METHOD M_Activity_Stop_PTCs : BOOL
VAR_INPUT
END_VAR
VAR_INST
	
END_VAR

out_bStop_PTCs := TRUE;

logs.M_LogInfo('STOP all PTCs...');
	
	
stat.nState := E_MET_CRYO_WARMUP_STATE.START_RAMP_Up_DETECTORS_1K;
END_METHOD

METHOD M_Activity_Stopping_Warm_Up
VAR_INPUT
END_VAR
VAR_IN_OUT
	{attribute 'OPC.UA.DA' := '0'}
	all_cryo_temps:					FB_METIS_TEMPERATURES;
	{attribute 'OPC.UA.DA' := '0'}
	all_heaters:					FB_METIS_HEATERS;
	{attribute 'OPC.UA.DA' := '0'}
	all_t_ctrls:      				FB_METIS_TCTRL;
	{attribute 'OPC.UA.DA' := '0'}
	all_t_votes: 					FB_METIS_VOTERS;
	{attribute 'OPC.UA.DA' := '0'}
	interlocks:						T_METIS_CRYO_INTERLOCKS;
END_VAR
// TODO CRY VOTE 8 



	all_heaters.h_cry_sha.M_SetDisable();
	all_heaters.h_cry_shb.M_SetDisable();
	all_heaters.h_cry_shc.M_SetDisable();

	all_t_ctrls.tc_cry_sha.M_SetDisable();
	all_t_ctrls.tc_cry_shb.M_SetDisable();
	all_t_ctrls.tc_cry_shc.M_SetDisable();
	stat.nState := E_MET_CRYO_WARMUP_STATE.FINISHED;
	stat.sState := 'Stopping Warm Up...';
	
	logs.M_LogInfo('Stopping heaters and temperature controls...');
END_METHOD

METHOD M_AreWarmUpHeaterActive : BOOL
VAR_INPUT
END_VAR
END_METHOD

METHOD M_CheckTCErrors
VAR_INPUT
END_VAR
VAR_IN_OUT
	{attribute 'OPC.UA.DA' := '0'}
	all_cryo_temps:					FB_METIS_TEMPERATURES;
	{attribute 'OPC.UA.DA' := '0'}
	all_heaters:					FB_METIS_HEATERS;
	{attribute 'OPC.UA.DA' := '0'}
	all_t_ctrls:      				FB_METIS_TCTRL;
	{attribute 'OPC.UA.DA' := '0'}
	all_t_votes: 					FB_METIS_VOTERS;
	{attribute 'OPC.UA.DA' := '0'}
	interlocks:						T_METIS_CRYO_INTERLOCKS;
END_VAR
IF all_heaters.h_cry_sha.M_isHeaterInError() OR all_t_ctrls.tc_cry_sha.stat.bError THEN
	stat.bError := TRUE;
	//M_SetError(E8100_StiffRingTempCtrlError, 'ERROR: Stiff Ring temp control - Check the complete Control-loop');

END_IF

IF all_heaters.h_cry_shb.M_isHeaterInError() OR all_t_ctrls.tc_cry_shb.stat.bError THEN
	stat.bError := TRUE;
	//M_SetError(E8101_IntermediateSegmentTempCtrlError, 'ERROR: Intermediate segment temp control - Check the complete Control-loop');
END_IF

IF all_heaters.h_cry_shc.M_isHeaterInError() OR all_t_ctrls.tc_cry_shc.stat.bError THEN
	stat.bError := TRUE;
	//M_SetError(E8102_BottomSegmentTempCtrlError, 'ERROR: Bottom Segment - Check the complete Control-loop');

END_IF

IF (all_heaters.h_cry_sha.M_isHeaterInError() OR all_t_ctrls.tc_cry_sha.stat.bError) AND 
	(all_heaters.h_cry_shb.M_isHeaterInError() OR all_t_ctrls.tc_cry_shb.stat.bError) AND
	(all_heaters.h_cry_shc.M_isHeaterInError() OR all_t_ctrls.tc_cry_shc.stat.bError) THEN
	stat.bError := TRUE;
	//M_SetError(E8103_OneOrMoreTempCtrlInError, 'ERROR: One or more temp control - Check the Control-loop');
	RETURN;
END_IF
END_METHOD

METHOD M_Configure
VAR_INPUT
END_VAR
IF NOT stat.bConfigured THEN


// Event Handleing 

arrEventEntry[0] := Tc_Events.METIS_Cryo_Routine.Routine_Started;
arrEventEntry[1] := Tc_Events.METIS_Cryo_Routine.Routine_Stopped_Manually;
arrEventEntry[2] := Tc_Events.METIS_Cryo_Routine.Routine_Stopped_Automatically;
arrEventEntry[3] := Tc_Events.METIS_Cryo_Routine.Routine_Completed_Successfully;
arrEventEntry[4] := Tc_Events.METIS_Cryo_Routine.Routine_FailedToStart;
arrEventEntry[5] := Tc_Events.METIS_Cryo_Routine.Routine_Aborted_CriticalFault;
arrEventEntry[6] := Tc_Events.METIS_Cryo_Routine.Routine_Interlock_ConflictDetected;


//////


// This call just configures logs at the very start.
// Logging is done by explicit calls to M_LogInfo().
logs(in_sName := in_sName);



// A MUST !!!
stat.bConfigured	:= TRUE;


END_IF
END_METHOD

METHOD M_HandleEvents
VAR_INPUT
END_VAR

//
// Handle triggers
//

trigEnable	(CLK := ctrl.bEnable);
trigDisable	(CLK := ctrl.bEnable);

// Array of EventEntry is initialised in the M_Configure method with 
// the alarms defined for the Valve.

fbAlarmHandler(stAlarms := stAlarms);


// Set Alarms

IF trigEnable.Q	THEN
	fbAlarmHandler.M_SetAlarm(Tc_Events.METIS_Cryo_Routine.Routine_Started);
END_IF

IF trigDisable.Q	THEN
	fbAlarmHandler.M_SetAlarm(Tc_Events.METIS_Cryo_Routine.Routine_Stopped_Manually);
END_IF

IF stat.bDone THEN
	fbAlarmHandler.M_SetAlarm(Tc_Events.METIS_Cryo_Routine.Routine_Completed_Successfully);
END_IF

IF stat.bAlarm THEN
	fbAlarmHandler.M_SetAlarm(Tc_Events.METIS_Cryo_Routine.Routine_Aborted_CriticalFault);
	fbAlarmHandler.M_SetAlarm(Tc_Events.METIS_Cryo_Routine.Routine_Stopped_Automatically);
END_IF

IF stat.bError THEN
	fbAlarmHandler.M_SetAlarm(Tc_Events.METIS_Cryo_Routine.Routine_FailedToStart);
END_IF

// Clear Alarms

IF NOT stat.bAlarm THEN
	fbAlarmHandler.M_ClearAlarm(Tc_Events.METIS_Cryo_Routine.Routine_Aborted_CriticalFault);
	fbAlarmHandler.M_ClearAlarm(Tc_Events.METIS_Cryo_Routine.Routine_Stopped_Automatically);
END_IF

IF NOT stat.bError THEN
	fbAlarmHandler.M_ClearAlarm(Tc_Events.METIS_Cryo_Routine.Routine_FailedToStart);
END_IF
END_METHOD

METHOD M_HandleInterlocks
VAR_INPUT
END_VAR
VAR_IN_OUT
	{attribute 'OPC.UA.DA' := '0'}
	all_cryo_temps:					FB_METIS_TEMPERATURES;
	{attribute 'OPC.UA.DA' := '0'}
	all_heaters:					FB_METIS_HEATERS;
	{attribute 'OPC.UA.DA' := '0'}
	all_t_ctrls:      				FB_METIS_TCTRL;
	{attribute 'OPC.UA.DA' := '0'}
	all_t_votes: 					FB_METIS_VOTERS;
	{attribute 'OPC.UA.DA' := '0'}
	interlocks:						T_METIS_CRYO_INTERLOCKS;
END_VAR



//interlocks.bInterlock_Evacuation 		:= FALSE;
//interlocks.bInterlock_Venting 			:= TRUE; // Venting blocked
//interlocks.bInterlock_CoolDown 			:= TRUE; // Cool_Down, pre-cooling, LN2_filling blocked
//interlocks.bInterlock_WarmUp 			:= TRUE; // Warm_up Blocked
//interlocks.bInterlock_Regeneration 		:= FALSE;
//interlocks.bInterlock_AntiFogging 		:= FALSE;
//interlocks.bInterlock_PowerOutage 		:= FALSE;
//interlocks.bInterlock_StopPowerOutage	:= FALSE;

//interlocks.sInterlockState := 'RE_GENERATION Active';
END_METHOD

METHOD M_PermitEvacuationStop : BOOL
VAR_INPUT
END_VAR
M_PermitEvacuationStop := stat.bPermitEvacuationStop;
END_METHOD

METHOD M_PermitVenting : BOOL
VAR_INPUT
END_VAR
END_METHOD

METHOD PRIVATE M_SetError
VAR_INPUT
    nCode     : UDINT;
    sMessage  : STRING;
END_VAR


stat.Error.nCode := nCode;
stat.Error.sMessage := sMessage;
stat.bError := TRUE;
//stat.nState := E_MET_CRYO_WARMUP_STATE.ERROR;
END_METHOD

METHOD M_StateMachine
VAR_INPUT
END_VAR
VAR_IN_OUT
	{attribute 'OPC.UA.DA' := '0'}
	all_cryo_temps:					FB_METIS_TEMPERATURES;
	{attribute 'OPC.UA.DA' := '0'}
	all_heaters:					FB_METIS_HEATERS;
	{attribute 'OPC.UA.DA' := '0'}
	all_t_ctrls:      				FB_METIS_TCTRL;
	{attribute 'OPC.UA.DA' := '0'}
	all_t_votes: 					FB_METIS_VOTERS;
	{attribute 'OPC.UA.DA' := '0'}
	interlocks:						T_METIS_CRYO_INTERLOCKS;
END_VAR


//--- State Machine Logic ---
CASE stat.nState OF
	
	E_MET_CRYO_WARMUP_STATE.NONE:
		
		M_Activity_None(interlocks := interlocks);
 
	E_MET_CRYO_WARMUP_STATE.CHECK_PRECONDITIONS:
	
		M_Activity_Check_Preconditions(); 
	
	E_MET_CRYO_WARMUP_STATE.START_WARM_UP:
	
		M_Activity_Start_Warm_Up();
		
	E_MET_CRYO_WARMUP_STATE.STOP_PTCs:
	
		M_Activity_Stop_PTCs();
 	
	E_MET_CRYO_WARMUP_STATE.START_RAMP_Up_DETECTORS_1K:
	
		M_Activity_Start_Ramp_Up_Detectors_1k();
	
	E_MET_CRYO_WARMUP_STATE.KEEP_RAMPING_Up_DETECTORS:
	
		M_Activity_Keep_Ramping_Up_Detectors();
	
	E_MET_CRYO_WARMUP_STATE.RAMP_UP_DETECTORS_6K:
	
		M_Activity_Ramp_Up_Detectors_2();
	
	E_MET_CRYO_WARMUP_STATE.START_RAMP_Up_RADIATION_SHIELDS:
	
		M_Activity_Start_Ramp_Up_Radiation_Shields(		
						all_cryo_temps:= all_cryo_temps,
						all_heaters := all_heaters,
						all_t_ctrls := all_t_ctrls,
						all_t_votes := all_t_votes,
						interlocks := interlocks);
		M_CheckTCErrors(all_cryo_temps:= all_cryo_temps,
						all_heaters := all_heaters,
						all_t_ctrls := all_t_ctrls,
						all_t_votes := all_t_votes,
						interlocks := interlocks);
	
	E_MET_CRYO_WARMUP_STATE.START_RAMP_Up_IMG:
	
		M_Activity_Start_Ramp_Up_IMG();
	
	E_MET_CRYO_WARMUP_STATE.START_RAMP_Up_SCAO:
	
		M_Activity_Start_Ramp_Up_SCAO();
	
	E_MET_CRYO_WARMUP_STATE.START_RAMP_Up_LMS:
	
		M_Activity_Start_Ramp_Up_LMS();
	
	E_MET_CRYO_WARMUP_STATE.START_RAMP_Up_CFO:
	
		M_Activity_Start_Ramp_Up_CFO();
	
	E_MET_CRYO_WARMUP_STATE.KEEP_WARMING_UP:
	
		M_Activity_Keep_Warming_Up(all_cryo_temps:= all_cryo_temps);
		
		M_CheckTCErrors(all_cryo_temps:= all_cryo_temps,
						all_heaters := all_heaters,
						all_t_ctrls := all_t_ctrls,
						all_t_votes := all_t_votes,
						interlocks := interlocks);
	
	E_MET_CRYO_WARMUP_STATE.STOPPING_WARM_UP:
	
		M_Activity_Stopping_Warm_Up(all_cryo_temps:= all_cryo_temps,
						all_heaters := all_heaters,
						all_t_ctrls := all_t_ctrls,
						all_t_votes := all_t_votes,
						interlocks := interlocks);
	
	E_MET_CRYO_WARMUP_STATE.FINISHED:
	
		M_Activity_Finished(); 
	
	E_MET_CRYO_WARMUP_STATE.ERROR:
	
		M_Activity_Error_Handling(all_cryo_temps:= all_cryo_temps,
						all_heaters := all_heaters,
						all_t_ctrls := all_t_ctrls,
						all_t_votes := all_t_votes,
						interlocks := interlocks);

END_CASE;
END_METHOD

METHOD M_UpdateStatus
VAR_INPUT
END_VAR


IF stat.nState = E_MET_CRYO_WARMUP_STATE.ERROR THEN
	stat.bError := TRUE;
ELSE
	stat.bError := FALSE;
END_IF



out_bWarmUpActive := stat.bActive;


// Check Pre-Conditions for HMI Enable 


stat.bPreConditionsMet := 	in_Cryo_Stat.bPumpsAreRunning 		AND
							in_Cryo_Stat.bEvacuationActive   	AND
							NOT in_Cryo_Stat.bCoolDownActive    AND
							in_Cryo_Stat.bVentingValvesAreClosed;
END_METHOD

END_FUNCTION_BLOCK

// POUs/Routines/Regeneration/FB_METIS_CRYO_REGENERATION
FUNCTION_BLOCK FB_METIS_CRYO_REGENERATION
VAR_INPUT
	in_sName:								STRING := 'RE-GENERATION';
	in_Cryo_Stat:							T_METIS_CRYO_STAT;
	in_lrRegeneration_Safe_Temp:			LREAL := 280.0;
	in_lrRegeneration_Safe_Press:			LREAL := 0.01;
    in_lrTemp_Regeneration_SetPoint: 		LREAL := 333.0;
    in_lrTemp_Regeneration_Alarm:			LREAL := 340.0;
    in_lrTemp_Regeneration_Stop:			LREAL := 310.0;
    in_tSorption_Pump_Cool_Down_TimeOut: 	TIME  := T#3H; 
END_VAR
VAR_OUTPUT
	out_bRegenerationActive : BOOL := FALSE; // TRUE when regeneration is active
END_VAR

VAR_IN_OUT
	{attribute 'OPC.UA.DA' := '0'}
	all_cryo_temps:					FB_METIS_TEMPERATURES;
	{attribute 'OPC.UA.DA' := '0'}
	all_heaters:					FB_METIS_HEATERS;
	{attribute 'OPC.UA.DA' := '0'}
	all_t_ctrls:      				FB_METIS_TCTRL;
	{attribute 'OPC.UA.DA' := '0'}
	all_t_votes: 					FB_METIS_VOTERS;
	{attribute 'OPC.UA.DA' := '0'}
	interlocks:						T_METIS_CRYO_INTERLOCKS;
END_VAR
VAR	
	t_vote_tc_cry_sp:				FB_METIS_VOTER;
	tc_sorption_pump:				FB_PWM_PID_CTRL;
	h_sorption_pump_heater:			FB_HEATER_PWM;		// 3.4 A terminal
	
	stat:							T_MET_CRYO_RE_GENERATION_STAT;
	ctrl:							T_MET_CRYO_RE_GENERATION_CTRL;


	
	bTest_run: BOOL := FALSE;
	
		// Triggers.
	//
	// Capture Enable/Disable.
	trigEnable:		R_TRIG;	// in_bEnable
	trigDisable:	F_TRIG;	// in_bEnable
	
	/////////////////////
	// Cryo System logs
	/////////////////////
		
	logs:	FB_CRYO_FUNCTION_LOG;
	
	// timeouts
	
	tonHeatingTimer     : TON;         // Timer to track the 3-hour heating period
	tHeatingTime:		TIME;
	lrHeatingTime:		LREAL := 3.0; // hours
	
	CoolDownTimeout:		TON;
	tCoolDownTime:			TIME;
	lrCoolDownTime:			LREAL := 1.0; // hours
	
	
END_VAR
VAR CONSTANT

    // --- [2000] Preconditions ---
    E2000_TemperaturesTooLow                      : UDINT := 2000001; // One or more cryostat temperatures < 280 K
    E2001_EvacuationNotActive                     : UDINT := 2000002; // Evacuation system not active
    E2002_RegenerationAlreadyRunning              : UDINT := 2000003; // Regeneration requested while already active
    E2003_CryostatPressureTooHigh_PreStart        : UDINT := 2000004; // Cryostat pressure > 1e-2 mbar before regeneration

    // --- [2100] Heater / Temperature Control Errors ---
    E2100_SorptionHeaterNotEnabled                : UDINT := 2100001; // Sorption pump heater failed to enable
    E2101_SorptionHeaterControlNotStarted         : UDINT := 2100002; // Temperature control did not start
    E2102_SorptionHeaterFailure                   : UDINT := 2100003; // Sorption pump heater failure detected
    E2103_SorptionHeaterShutdownFailure           : UDINT := 2100004; // Heater did not stop after regeneration

    // --- [2200] Temperature Monitoring Errors ---
    E2200_SP_TemperatureSensorFault               : UDINT := 2200001; // Sorption pump temperature sensor invalid
    E2201_SP_TemperatureNotRising                 : UDINT := 2200002; // Temperature not increasing during heating
    E2202_SP_TemperatureTooHigh                   : UDINT := 2200003; // Sorption pump temperature > 340 K
    E2203_SP_TemperatureNotCooling                : UDINT := 2200004; // Sorption pump not cooling after heater shutdown
    E2204_SP_CooldownTimeout                      : UDINT := 2200005; // Sorption pump cooldown timeout exceeded

    // --- [2300] Pressure Monitoring Errors ---
    E2300_CryostatPressureTooHigh                 : UDINT := 2300001; // Cryostat pressure > 1e-2 mbar during regeneration
    E2301_CryostatPressureRiseUnexpected          : UDINT := 2300002; // Unexpected pressure increase detected

    // --- [2400] Sequence Timing Errors ---
    E2400_RegenerationHeatingTimeout              : UDINT := 2400001; // Temperature did not reach target within allowed time
    E2401_RegenerationHoldTimeNotCompleted        : UDINT := 2400002; // 3-hour heating hold interrupted
    E2402_RegenerationSequenceTimeout             : UDINT := 2400003; // Regeneration procedure exceeded maximum duration

    // --- [2500] Manual Intervention ---
    E2500_OperatorStoppedRegeneration             : UDINT := 2500001; // Operator manually stopped regeneration
    E2501_OperatorDisabledHeater                  : UDINT := 2500002; // Heater disabled manually during regeneration

    // --- [2600] Interlock Violations ---
    E2600_LN2FillingActiveDuringRegeneration      : UDINT := 2600001; // Vessel filling active during regeneration
    E2601_PrecoolingActiveDuringRegeneration      : UDINT := 2600002; // Precooling system active during regeneration
    E2602_VentingActiveDuringRegeneration         : UDINT := 2600003; // Venting active during regeneration
    E2603_CoolingActiveDuringRegeneration         : UDINT := 2600004; // Cooling routine active during regeneration

    // --- [2700] Shutdown / Recovery Failures ---
    E2700_HeaterDidNotDisable                     : UDINT := 2700001; // Heater failed to disable during shutdown
    E2701_TemperatureControlDidNotStop            : UDINT := 2700002; // Temperature control still active after stop command
    E2702_RegenerationShutdownTimeout             : UDINT := 2700003; // Regeneration shutdown timeout exceeded

END_VAR


(*
	TODO: One of the initial conditions checks the minimum temperatures in the cryostat.
	The is still an open question to how to determine that.
	For time being with empty cryostat, a temperature on the Cryo body is considered to check the 
	minimum temperature 
*)

M_Configure();

M_HandleEvents();

M_ExecuteControllers();

M_StateMachine( 
	all_cryo_temps:= 							all_cryo_temps, 
	all_heaters:= 								all_heaters, 
	all_t_ctrls:= 								all_t_ctrls, 
	all_t_votes:=								all_t_votes, 
	interlocks:= 								interlocks);

M_UpdateStatus();



tHeatingTime := LREAL_TO_TIME(lrHeatingTime *  3600000.0);
tCoolDownTime := LREAL_TO_TIME(lrCoolDownTime * 3600000.0);

(* Re-Generation *)
METHOD M_Activity_Check_Preconditions : BOOL
VAR_INPUT
END_VAR
VAR_IN_OUT
	{attribute 'OPC.UA.DA' := '0'}
	all_cryo_temps:					FB_METIS_TEMPERATURES;
	{attribute 'OPC.UA.DA' := '0'}
	all_heaters:					FB_METIS_HEATERS;
	{attribute 'OPC.UA.DA' := '0'}
	all_t_ctrls:      				FB_METIS_TCTRL;
	{attribute 'OPC.UA.DA' := '0'}
	all_t_votes: 					FB_METIS_VOTERS;
	{attribute 'OPC.UA.DA' := '0'}
	interlocks:						T_METIS_CRYO_INTERLOCKS;
END_VAR


//  Precondition Check: Cryo Temperature validity
IF NOT in_Cryo_Stat.bLowestTempValid THEN
	//M_SetError(nCode := E3101_REGEN_INVALID_TEMP,
	//			sMessage := 'Error: Invalid lowest cryo temperature reading.');
	stat.sRecoverySuggestion := '';
	RETURN; 
END_IF

//  Precondition Check: Regeneration safe Temperature 
IF in_Cryo_Stat.lrLowestTempK <= in_lrRegeneration_Safe_Temp THEN

	stat.sState := 'Error: temperature is below the safe Regeneration temperature.';
	//M_SetError(nCode := E3107_REGEN_SYSTEM_BELOW_SAFE_REGEN,
	//			sMessage := 'Error: system temperature is below the safe Regeneration temp.');
	stat.sRecoverySuggestion := '';
	RETURN; // Exit this state
END_IF


//  Precondition Check: Evacuation Status 
IF NOT in_Cryo_Stat.bEvacuationActive THEN

	stat.nState := E_MET_CRYO_RE_GENERATION_STATE.CHECK_PRECONDITIONS;
	///M_SetError(nCode := E3108_REGEN_EVACUATION_NOT_ACTIVE,
	//			sMessage := 'Error: Evacuation not Active');
		stat.sRecoverySuggestion := 'Start Evacuation';			
	stat.bPermitEvacuationStop := FALSE; // Prevent premature stop of evacuation
	RETURN; // Exit this state until evacuation is active
END_IF

{IF defined (V1_HW)}

//  Precondition Check: Evacuation Status 
IF NOT in_Cryo_Stat.bRoughingPumpsAreRunning THEN

	stat.nState := E_MET_CRYO_RE_GENERATION_STATE.CHECK_PRECONDITIONS;
	M_SetError(nCode := E3106_REGEN_PUMPS_NOT_ACTIVE,
				sMessage := 'Error: One or both roughing pumps are not running');
		stat.sRecoverySuggestion := 'Start roughing pumps';			
	stat.bPermitEvacuationStop := FALSE; // Prevent premature stop of evacuation
	RETURN; // Exit this state until evacuation is active
	
ELSE
	
		;
END_IF

{END_IF}

stat.bActive := TRUE;
stat.bBusy 	 := TRUE;
stat.bDone   := FALSE;

// If all preconditions are met, proceed to the next state
stat.nState := E_MET_CRYO_RE_GENERATION_STATE.START_HEATING;

stat.sState := 'Regenerating...';
logs.M_LogInfo('Regeneration Started...');
END_METHOD

METHOD M_Activity_CoolDownSP : BOOL
VAR_INPUT
END_VAR
VAR_IN_OUT
	{attribute 'OPC.UA.DA' := '0'}
	all_cryo_temps:					FB_METIS_TEMPERATURES;
	{attribute 'OPC.UA.DA' := '0'}
	all_heaters:					FB_METIS_HEATERS;
	{attribute 'OPC.UA.DA' := '0'}
	all_t_ctrls:      				FB_METIS_TCTRL;
	{attribute 'OPC.UA.DA' := '0'}
	all_t_votes: 					FB_METIS_VOTERS;
	{attribute 'OPC.UA.DA' := '0'}
	interlocks:						T_METIS_CRYO_INTERLOCKS;
END_VAR
	all_heaters.h_cry_sp.M_SetDisable();
	all_t_ctrls.tc_cry_sp.M_SetDisable();
	tonHeatingTimer(IN:=FALSE); // Reset Timer
	
	IF all_cryo_temps.t_cry_vot_10.stat.lrTempK < in_lrTemp_Regeneration_Stop THEN
		stat.nState := E_MET_CRYO_RE_GENERATION_STATE.FINISHED;
		cooldownTimeout(IN := FALSE);
	ELSE
		stat.nState := E_MET_CRYO_RE_GENERATION_STATE.COOL_DOWN;
		stat.sState := 'Sorption-pump cooling down';
	END_IF
	
	cooldownTimeout(IN := TRUE, PT := tCoolDownTime);
	stat.sState :=  CONCAT('Sorption-pump cooling down...', F_TON_TO_TIME_STRING(Timer := cooldownTimeout));

	IF cooldownTimeout.Q THEN
		logs.M_LogWarning('Cooldown timeout. Sorption pump did not cool sufficiently.');
		cooldownTimeout(IN := FALSE);
		//stat.nState := E_MET_CRYO_RE_GENERATION_STATE.ERROR;
		RETURN;
	END_IF
END_METHOD

METHOD M_Activity_ErrorHandeling : BOOL
VAR_INPUT
END_VAR
VAR_IN_OUT
	{attribute 'OPC.UA.DA' := '0'}
	all_cryo_temps:					FB_METIS_TEMPERATURES;
	{attribute 'OPC.UA.DA' := '0'}
	all_heaters:					FB_METIS_HEATERS;
	{attribute 'OPC.UA.DA' := '0'}
	all_t_ctrls:      				FB_METIS_TCTRL;
	{attribute 'OPC.UA.DA' := '0'}
	all_t_votes: 					FB_METIS_VOTERS;
	{attribute 'OPC.UA.DA' := '0'}
	interlocks:						T_METIS_CRYO_INTERLOCKS;
END_VAR
        stat.bActive := TRUE;
        in_cryo_stat.bPermitEvacuationStop := FALSE; // Evacuation cannot stop, yet
		all_heaters.h_cry_sp.M_SetDisable();
		all_t_ctrls.tc_cry_sp.M_SetDisable();
        
		IF all_cryo_temps.t_cry_vot_10.stat.lrTempK < in_lrTemp_Regeneration_Stop THEN
            stat.nState := E_MET_CRYO_RE_GENERATION_STATE.NONE;
			stat.bActive := FALSE;
			stat.bBusy := FALSE;
			ctrl.bEnable := FALSE;						// Disable Regeneration
			stat.bPermitEvacuationStop := TRUE; // Evacuation can stop
		ELSE
			stat.nState := E_MET_CRYO_RE_GENERATION_STATE.COOL_DOWN;
			stat.sState := 'Sorption-pump cooling down';
        END_IF
		
        IF ctrl.bReset THEN
			logs.M_LogInfo('Reset received. Restarting regeneration.'); 
            stat.nState := E_MET_CRYO_RE_GENERATION_STATE.NONE;
			ctrl.bReset := FALSE;
			ctrl.bEnable := FALSE;						// Disable Regeneration
        END_IF
END_METHOD

METHOD M_Activity_Finished : BOOL
VAR_INPUT
END_VAR
VAR_IN_OUT
	{attribute 'OPC.UA.DA' := '0'}
	all_cryo_temps:					FB_METIS_TEMPERATURES;
	{attribute 'OPC.UA.DA' := '0'}
	all_heaters:					FB_METIS_HEATERS;
	{attribute 'OPC.UA.DA' := '0'}
	all_t_ctrls:      				FB_METIS_TCTRL;
	{attribute 'OPC.UA.DA' := '0'}
	all_t_votes: 					FB_METIS_VOTERS;
	{attribute 'OPC.UA.DA' := '0'}
	interlocks:						T_METIS_CRYO_INTERLOCKS;
END_VAR


//stat.bPermitEvacuationStop := TRUE; // Evacuation can stop
all_heaters.h_cry_sp.M_SetDisable();
all_t_ctrls.tc_cry_sp.M_SetDisable();
stat.sState := 'Re_generation finished';
tonHeatingTimer.IN := FALSE; // Reset Timer
	
ctrl.bEnable := FALSE;			// Disable Regeneration

stat.nState := E_MET_CRYO_RE_GENERATION_STATE.NONE;
logs.M_LogInfo('Sorption regeneration finished.');

stat.bActive := FALSE;
stat.bBusy 	 := FALSE;
stat.bDone   := TRUE;

cooldownTimeout(IN := FALSE);
tonHeatingTimer(IN := FALSE);
END_METHOD

METHOD M_Activity_KeepHeating : BOOL
VAR_INPUT
END_VAR
VAR_IN_OUT
    {attribute 'OPC.UA.DA' := '0'}
    all_cryo_temps : FB_METIS_TEMPERATURES;
    {attribute 'OPC.UA.DA' := '0'}
    all_heaters    : FB_METIS_HEATERS;
    {attribute 'OPC.UA.DA' := '0'}
    all_t_ctrls    : FB_METIS_TCTRL;
    {attribute 'OPC.UA.DA' := '0'}
    all_t_votes    : FB_METIS_VOTERS;
    {attribute 'OPC.UA.DA' := '0'}
    interlocks     : T_METIS_CRYO_INTERLOCKS;
END_VAR
VAR_INST
    nHeatingState  : UINT := 0;
    bLoggedReached : BOOL := FALSE;
	
	tonTempSenseGlitch : TON;                 // 3 minute grace window
    bTempSenseGlitchActive : BOOL := FALSE;   // latched while in grace window
END_VAR
VAR
    lrTempK        : LREAL;
    bHeaterError   : BOOL;
    bOverTemp      : BOOL;
    bDisableReq    : BOOL;

    bTempGlitchNow  : BOOL;
END_VAR
M_Activity_KeepHeating := FALSE;

// Snapshot values
lrTempK      := all_cryo_temps.t_cry_vot_10.stat.lrTempK;
bHeaterError := all_heaters.h_cry_sp.M_isHeaterInError();
bDisableReq  := trigDisable.Q;

////////////////////////////////////////////////////
// Temp Sensor glitch handling: lrTempK forced to >900K
////////////////////////////////////////////////////
bTempGlitchNow := (lrTempK > 900.0);

// Start / run 3-minute grace timer while glitch is present
IF bTempGlitchNow THEN
    bTempSenseGlitchActive := TRUE;
    tonTempSenseGlitch(IN := TRUE, PT := T#3M);

ELSE
    // Glitch not present now
    IF bTempSenseGlitchActive THEN
        // We were in a glitch window and it recovered before timing out
        IF NOT tonTempSenseGlitch.Q THEN
            //M_SetError(E3000_REGEN_ERROR_CLEARED, '');
            stat.sRecoverySuggestion := '';
        END_IF

        // Stop and reset the glitch timer/window
        bTempSenseGlitchActive := FALSE;
        tonTempSenseGlitch(IN := FALSE, PT := T#3M);
    ELSE
        // Ensure timer is reset if not used
        tonTempSenseGlitch(IN := FALSE, PT := T#3M);
    END_IF
END_IF

// If glitch persists beyond 3 minutes, we stop masking.
// From that moment onward, the normal over-temperature check may act.
IF bTempSenseGlitchActive AND tonTempSenseGlitch.Q THEN
    // Grace window expired -> stop masking further
    bTempSenseGlitchActive := FALSE;
    tonTempSenseGlitch(IN := FALSE, PT := T#3M);
END_IF

//////////////////////////////////////////
// operator interrupt / errors
/////////////////////////////////////////

// Operator interrupt
IF bDisableReq THEN
    stat.sState := 'REGENERATION interrupted by the operator...';
    logs.M_LogInfo('REGENERATION interrupted by the operator...');
    stat.nState := E_MET_CRYO_RE_GENERATION_STATE.COOL_DOWN;

    all_heaters.h_cry_sp.M_SetDisable();
    all_t_ctrls.tc_cry_sp.M_SetDisable();
    tonHeatingTimer(IN := FALSE);
    cooldownTimeout(IN := FALSE);

    // Reset internal state
    nHeatingState := 0;
    bLoggedReached := FALSE;

    // Reset EMI logic state too
    bTempSenseGlitchActive := FALSE;
    tonTempSenseGlitch(IN := FALSE, PT := T#3M);

    RETURN;
END_IF

// Over-temperature alarm: take action immediately,
// BUT only if we are NOT currently masking due to Temp Sensor glitch grace window.
bOverTemp := (lrTempK > in_lrTemp_Regeneration_Alarm);

IF bOverTemp AND (NOT bTempSenseGlitchActive) THEN
    logs.M_LogWarning('Temperature exceeds safe limit!');
    //M_SetError(E3102_REGEN_OVER_TEMP, 'Temperature at SP above alarm limit');
    stat.bAlarm := TRUE;

    stat.nState := E_MET_CRYO_RE_GENERATION_STATE.COOL_DOWN;
    stat.sState := 'Alarm: Sorption pump overheated';

    all_heaters.h_cry_sp.M_SetDisable();
    all_t_ctrls.tc_cry_sp.M_SetDisable();
    tonHeatingTimer(IN := FALSE);
    cooldownTimeout(IN := FALSE);

    // Reset internal state
    nHeatingState := 0;
    bLoggedReached := FALSE;

    // Reset Glitch logic state too
    bTempSenseGlitchActive := FALSE;
    tonTempSenseGlitch(IN := FALSE, PT := T#3M);

    RETURN;
END_IF

// Heater error 
IF all_heaters.h_cry_sp.M_isHeaterInError() THEN
{IF defined (V1_HW)}
 //   stat.nState := E_MET_CRYO_RE_GENERATION_STATE.COOL_DOWN;
    logs.M_LogInfo('SP heater failed, Regeneration stopped.');
    stat.sState := 'Heater error';
    M_SetError(E3105_REGEN_HEATER_FAIL, 'Heater at SP failed');
    stat.sRecoverySuggestion := 'Check SP heater controller';

//    all_heaters.h_cry_sp.M_SetDisable();
//    all_t_ctrls.tc_cry_sp.M_SetDisable();
//    tonHeatingTimer(IN := FALSE);
//    cooldownTimeout(IN := FALSE);

//    // Reset internal state
//    nHeatingState := 0;
//    bLoggedReached := FALSE;

//    // Reset Glitch logic state too
//    bTempSenseGlitchActive := FALSE;
//    tonTempSenseGlitch(IN := FALSE, PT := T#3M);

    RETURN;
{END_IF}
END_IF

/////////////////////////////////////////////////////
// state machine (normal operation)
/////////////////////////////////////////////////////
CASE nHeatingState OF
    0:
        in_cryo_stat.sState := 'REGENERATION Active';
        stat.sState := CONCAT('Sorption pump heating up to ',
                       CONCAT(LREAL_TO_STRING(in_lrTemp_Regeneration_SetPoint), ' K'));

        tonHeatingTimer(IN := FALSE);

        IF lrTempK >= in_lrTemp_Regeneration_SetPoint THEN
            nHeatingState := 10;
            bLoggedReached := FALSE;
        END_IF

    10:
        IF NOT bLoggedReached THEN
            logs.M_LogInfo(CONCAT(LREAL_TO_STRING(in_lrTemp_Regeneration_SetPoint), ' K achieved at Sorption Pump'));
            bLoggedReached := TRUE;
        END_IF

        tonHeatingTimer(IN := TRUE, PT := tHeatingTime);

        stat.sState := CONCAT(
            'Sorption pump heating hold... ',
            F_TON_TO_TIME_STRING(Timer := tonHeatingTimer)
        );

        IF tonHeatingTimer.Q THEN
            tonHeatingTimer(IN := FALSE);
            nHeatingState := 20;
        END_IF

    20:
        stat.nState := E_MET_CRYO_RE_GENERATION_STATE.COOL_DOWN;
        stat.sState := 'Transition: heating duration completed';
        logs.M_LogWarning('Transition: heating duration completed');
        nHeatingState := 99;

    99:
        tonHeatingTimer(IN := FALSE);
        cooldownTimeout(IN := FALSE);
        nHeatingState := 0;
        bLoggedReached := FALSE;

    ELSE
        tonHeatingTimer(IN := FALSE);
        cooldownTimeout(IN := FALSE);
        nHeatingState := 0;
        bLoggedReached := FALSE;
END_CASE
END_METHOD

METHOD M_Activity_None : BOOL
VAR_INPUT
END_VAR
VAR_IN_OUT
	{attribute 'OPC.UA.DA' := '0'}
	all_cryo_temps:					FB_METIS_TEMPERATURES;
	{attribute 'OPC.UA.DA' := '0'}
	all_heaters:					FB_METIS_HEATERS;
	{attribute 'OPC.UA.DA' := '0'}
	all_t_ctrls:      				FB_METIS_TCTRL;
	{attribute 'OPC.UA.DA' := '0'}
	all_t_votes: 					FB_METIS_VOTERS;
	{attribute 'OPC.UA.DA' := '0'}
	interlocks:						T_METIS_CRYO_INTERLOCKS;
END_VAR
stat.bActive := FALSE;
stat.bBusy := FALSE;
stat.bDone := TRUE;
stat.bReadyToDisable := FALSE;
stat.bPermitEvacuationStop := FALSE; // Evacuation is not allowed to stop
tonHeatingTimer(IN:=FALSE, PT:= tHeatingTime);
cooldownTimeout(IN := FALSE);


IF ctrl.bEnable AND NOT interlocks.bInterlock_Regeneration THEN  // Check interlocks
	stat.nState := E_MET_CRYO_RE_GENERATION_STATE.CHECK_PRECONDITIONS;
	stat.sState := 'Starting...Checking Preconditions';
	logs.M_LogInfo('REGENERATION started by the operator...Checking Preconditions');
ELSE
	stat.nState := E_MET_CRYO_RE_GENERATION_STATE.NONE;
	stat.sState := 'Re_generation OFF';
END_IF
END_METHOD

METHOD M_Activity_StartHeating : BOOL
VAR_INPUT
END_VAR
VAR_IN_OUT
	{attribute 'OPC.UA.DA' := '0'}
	all_cryo_temps:					FB_METIS_TEMPERATURES;
	{attribute 'OPC.UA.DA' := '0'}
	all_heaters:					FB_METIS_HEATERS;
	{attribute 'OPC.UA.DA' := '0'}
	all_t_ctrls:      				FB_METIS_TCTRL;
	{attribute 'OPC.UA.DA' := '0'}
	all_t_votes: 					FB_METIS_VOTERS;
	{attribute 'OPC.UA.DA' := '0'}
	interlocks:						T_METIS_CRYO_INTERLOCKS;
END_VAR
        stat.bActive := TRUE;
		in_cryo_stat.sState := 'RE_GENERATION Active';
		
		stat.bPermitEvacuationStop := FALSE; // Evacuation is not allowed to stop
		
		// Enable SP Heater
		all_heaters.h_cry_sp.M_SetEnable();
		
		all_t_ctrls.tc_cry_sp.M_SetEnable();
		
		all_t_ctrls.tc_cry_sp.M_Set_SetPoint(
			m_eSetpointType := E_METIS_CTRL_SETPOINT_SWITCH.FIXED,
			m_lrFixedSetpoint := in_lrTemp_Regeneration_SetPoint,
			m_lrSetpointOffset := 0.0, 
			m_pSetpointTemp := all_cryo_temps.M_SetTemperatureSensor(0));
			
        tonHeatingTimer(IN:=TRUE, PT:= tHeatingTime);
		
        stat.nState := E_MET_CRYO_RE_GENERATION_STATE.KEEP_HEATING;
END_METHOD

METHOD M_Configure
VAR_INPUT
END_VAR

IF NOT stat.bConfigured THEN
	

// This call just configures logs at the very start.
// Logging is done by explicit calls to M_LogInfo().
logs(in_sName := in_sName);


stat.bConfigured := TRUE;

END_IF
END_METHOD

METHOD M_ExecuteControllers
VAR_INPUT
END_VAR





//h_sorption_pump_heater(in_sName:= , in_fHeaterResistance:= , in_nMaxHeaterPower:= , in_HeaterCtrlType:= );

//t_vote_tc_cry_sp(
//		in_sName:= 't_vote_tc_cry_sp', 
//		in_bSimulation:= FALSE, 
//		in_nRampPeriodSec:= 10, 
//		met_temp:= all_cryo_temps);
		
//tc_sorption_pump(
//	in_sName:= 'tc_sorption_pump',
//	in_bEnable:= ctrl.bEnable_Temp_Ctrl, 
//	in_lrSetPoint:= lrTemp_Regeneration_SetPoint,
//	heater:= h_sorption_pump_heater,
//	temperature:= t_vote_tc_cry_sp);
END_METHOD

METHOD M_HandleEvents
VAR_INPUT
END_VAR

//
// Handle triggers
//

trigEnable	(CLK := ctrl.bEnable);
trigDisable	(CLK := ctrl.bEnable);
END_METHOD

METHOD M_PermitEvacuationStop : BOOL
VAR_INPUT
END_VAR
M_PermitEvacuationStop := stat.bPermitEvacuationStop;
END_METHOD

METHOD PRIVATE M_SetError
VAR_INPUT
    nCode     : UDINT;
    sMessage  : STRING;
END_VAR


stat.Error.nCode := nCode;
stat.Error.sMessage := sMessage;
stat.bError := TRUE;
//stat.nState := E_MET_CRYO_RE_GENERATION_STATE.ERROR;
END_METHOD

METHOD M_StateMachine
VAR_INPUT
	
END_VAR
VAR_IN_OUT
	{attribute 'OPC.UA.DA' := '0'}
	all_cryo_temps:					FB_METIS_TEMPERATURES;
	{attribute 'OPC.UA.DA' := '0'}
	all_heaters:					FB_METIS_HEATERS;
	{attribute 'OPC.UA.DA' := '0'}
	all_t_ctrls:      				FB_METIS_TCTRL;
	{attribute 'OPC.UA.DA' := '0'}
	all_t_votes: 					FB_METIS_VOTERS;
	{attribute 'OPC.UA.DA' := '0'}
	interlocks:						T_METIS_CRYO_INTERLOCKS;
END_VAR
VAR_INST
		

END_VAR

CASE stat.nState OF
    E_MET_CRYO_RE_GENERATION_STATE.NONE:
	
		M_Activity_None(
				all_cryo_temps:= all_cryo_temps,
				all_heaters := all_heaters,
				all_t_ctrls := all_t_ctrls,
				all_t_votes := all_t_votes,
				interlocks := interlocks);

    E_MET_CRYO_RE_GENERATION_STATE.CHECK_PRECONDITIONS:

		M_Activity_Check_Preconditions(
				all_cryo_temps:= all_cryo_temps,
				all_heaters := all_heaters,
				all_t_ctrls := all_t_ctrls,
				all_t_votes := all_t_votes,
				interlocks := interlocks);
		
    E_MET_CRYO_RE_GENERATION_STATE.START_HEATING:
	
		M_Activity_StartHeating(
				all_cryo_temps:= all_cryo_temps,
				all_heaters := all_heaters,
				all_t_ctrls := all_t_ctrls,
				all_t_votes := all_t_votes,
				interlocks := interlocks);

	E_MET_CRYO_RE_GENERATION_STATE.KEEP_HEATING:
	
		M_Activity_KeepHeating(
				all_cryo_temps:= all_cryo_temps,
				all_heaters := all_heaters,
				all_t_ctrls := all_t_ctrls,
				all_t_votes := all_t_votes,
				interlocks := interlocks);
		
    E_MET_CRYO_RE_GENERATION_STATE.COOL_DOWN:
	
		M_Activity_CoolDownSP(
				all_cryo_temps:= all_cryo_temps,
				all_heaters := all_heaters,
				all_t_ctrls := all_t_ctrls,
				all_t_votes := all_t_votes,
				interlocks := interlocks);

    E_MET_CRYO_RE_GENERATION_STATE.FINISHED:
	
		M_Activity_Finished(
				all_cryo_temps:= all_cryo_temps,
				all_heaters := all_heaters,
				all_t_ctrls := all_t_ctrls,
				all_t_votes := all_t_votes,
				interlocks := interlocks);

    E_MET_CRYO_RE_GENERATION_STATE.ERROR:
	
		M_Activity_ErrorHandeling(
				all_cryo_temps:= all_cryo_temps,
				all_heaters := all_heaters,
				all_t_ctrls := all_t_ctrls,
				all_t_votes := all_t_votes,
				interlocks := interlocks);
	
END_CASE;
END_METHOD

METHOD M_UpdateStatus
VAR_INPUT
END_VAR


IF stat.nState = E_MET_CRYO_RE_GENERATION_STATE.ERROR THEN
	stat.bError := TRUE;
ELSE
	stat.bError := FALSE;
END_IF



out_bRegenerationActive := stat.bActive;

// Check Pre-Conditions for HMI Enable 

{IF defined (V1_HW)}

stat.bPreConditionsMet :=	in_Cryo_Stat.bRoughingPumpsAreRunning AND
							(in_Cryo_Stat.lrLowestTempK >= in_lrRegeneration_Safe_Temp);
{END_IF}
 


{IF defined (V2_SIM)}
stat.bPreConditionsMet :=	in_Cryo_Stat.bEvacuationActive AND
							(in_Cryo_Stat.lrLowestTempK >= in_lrRegeneration_Safe_Temp);

{END_IF}
END_METHOD

END_FUNCTION_BLOCK

// POUs/Control/Control/FB_PWM_PID_CTRL
FUNCTION_BLOCK FB_PWM_PID_CTRL EXTENDS FB_METIS_CTRL_BASE
VAR_INPUT
		//in_Temperature:	LREAL;
END_VAR
VAR_IN_OUT
	heater		:	FB_HEATER_PWM;
	temperature:	FB_METIS_VOTER;
END_VAR
VAR_OUTPUT
END_VAR
VAR
	
	bHeaterEnabled : 	BOOL := FALSE;
END_VAR


IF temperature.bTempValid THEN
	(* Set Actual value for PID *)
	//lrActualValue := in_Temperature;
	lrActualValue := temperature.lrTempK;
ELSIF temperature.bTempNotValid THEN
	(*If temp is not valid deactivate PID control*)
	eMode := eCTRL_MODE_MANUAL;

END_IF	




IF heater.bIsNotActive THEN
	heater.M_Activate();
ELSIF heater.bIsActive AND stat.bError THEN 
	heater.M_DeActivate();
END_IF



IF bEngMode THEN
	heater.M_SetManualInputFlag(TRUE);
ELSE
	heater.M_SetManualInputFlag(FALSE);
END_IF

 
	
SUPER^();

// Setting Power to the heater
IF bEngMode AND (NOT ctrl.bEnable) THEN
	lrControllerOut := lrManualOut; // set manual power
ELSE
	lrManualOut := lrControllerOut; // Bumpless transition
END_IF


//heater.M_GetHeaterPower(m_lrHeaterPower := lrControllerOut);

heater.lrHeaterPower := lrControllerOut;

END_FUNCTION_BLOCK

// POUs/Control/Control/FB_METIS_CTRL_BASE
FUNCTION_BLOCK FB_METIS_CTRL_BASE
VAR_INPUT
	in_sName:					STRING	;
	in_bEnable:					BOOL 	:= FALSE; 	// FALSE := manual control; TRUE := PID control active	
	in_lrSetPoint:				LREAL	;			//
	//in_lrRampUPRate:			LREAL 	;	// 1 Unit/min ramp-up (For warm-up)		
	//in_lrRampDownRate:			LREAL 	;	// 1 Unit/min ramp-Down (For Cool-down)

END_VAR
VAR_OUTPUT
END_VAR
VAR
	bAutoMode:					BOOL := TRUE;	// AUTO=true, MANUAL=false
	bManualMode:				BOOL := FALSE;	// Manual Mode
	bEngMode:					BOOL := FALSE;	// Commissioning/Engineering mode. Ignores interlocks
	
	bAutoModePermissions:		BOOL := TRUE;
	bManualModePermissions:		BOOL := FALSE;
	bEngModePermissions:		BOOL := FALSE;
	
	ctrl: 						T_METIS_CTRL_BASE_CTRL;
	stat: 						T_METIS_CTRL_BASE_STAT;
	cfg:						T_METIS_CTRL_BASE_CFG;
	
	(*Read/Write configuration*)
	
	fbTcConfig:				FB_READ_WRITE_TEMP_CONTROL_CONFIG;
	bReadConfig:			BOOL;
	bWriteConfig:			BOOL;
	(*Ramp control*)
	ramp:		FB_METIS_CTRL_RAMP_GENERATOR;
	
	lrRampSetpointValue				: LREAL		:= 330;
	(*PID Control*)
	
	lrSetpointValue					: LREAL; (* Output value from Ramp*)
	lrActualValue					: LREAL;
	lrManSyncValue					: LREAL;
	bSync							: BOOL;

	lrControllerOut					: LREAL;
	bHold							: BOOL;

	eMode							: E_CTRL_MODE;
	stCTRL_PID_PARAMS				: ST_CTRL_PID_PARAMS;

	eErrorId						: E_CTRL_ERRORCODES;
	bError							: BOOL;
	bARWactive						: BOOL;
	
	lrManualOut:		LREAL; // Input from HMI

	(* controller *)
	fbCTRL_PID						: FB_CTRL_PID;

	bInit							: BOOL	:= TRUE; 
	fbTON							: TON;
	
	(*Simulated Heating process to Generate ActualValue*)
	bSimulated					: BOOL := FALSE;					
	sim_heating_process			: FB_FT1_SIM_PROCESS;
		
END_VAR


(*Read/Write configuration*)
fbTcConfig(in_sTempCtrlName:= in_sName, Temp_Ctrl_Config:= cfg);


(*Configure*)
M_Configure();

M_SetPermissionMode();

(*Ramp control*)

//M_SetRamp(m_fSetPoint := in_fSetPoint, m_fRampUPRate := in_fRampUPRate, m_fRampDownRate := in_fRampDownRate);
M_SetRamp();

M_Set_PID_Parameters();

M_CheckErrors();

(*Execute PID controller*)

M_ExecuteController();



(* generate input signal *)
	fbTON(		IN:= TRUE,
				PT:= T#30S
			);
	IF fbTON.Q
	THEN
		fbTON(		IN:= FALSE);
		//fSetpointValue := -1.0 * fSetpointValue;
		lrRampSetpointValue := 0;
	END_IF

(* copy var to scope var *)
//fSetpointValueToScope 	:= fSetpointValue;
//fActualValueToScope 		:= fActualValue;



(*Simulated Heating process to Generate ActualValue*)
IF bSimulated THEN

	sim_heating_process(fIn:= lrControllerOut, fOut=> lrActualValue);

END_IF

METHOD M_CheckErrors : BOOL
VAR_INPUT
END_VAR
END_METHOD

METHOD M_Configure : BOOL
VAR_INPUT
END_VAR


IF NOT stat.bConfigured	THEN

fbTcConfig.M_ReadConfiguration();


(* init parameter struct *)
	stCTRL_PID_PARAMS.tCtrlCycleTime		:= T#10ms;
	stCTRL_PID_PARAMS.tTaskCycleTime		:= T#10ms;

	stCTRL_PID_PARAMS.fOutMaxLimit			:= 100.0;		(* maximum output limit				*)
	stCTRL_PID_PARAMS.fOutMinLimit			:= 0.0;			(* minimum output limit				*)

	(* set the mode to MANUAL --> Initialize with manual operation before PID is activated*)
	eMode							:= eCTRL_MODE_MANUAL;

	stat.bConfigured	:= TRUE;;
ELSE
	RETURN;	// Nothing to do any more
END_IF
END_METHOD

METHOD M_ExecuteController : BOOL
VAR_INPUT
END_VAR


(*
IF some condition THEN
Chnage the mode of PID to :

eMode := eCTRL_MODE_ACTIVE;
eMode := eCTRL_MODE_IDLE;
eMode := eCTRL_MODE_MANUAL;
eMode := eCTRL_MODE_RESET;

*)



(* call controller *)
fbCTRL_PID(		fSetpointValue			:= lrSetpointValue,
					fActualValue		:= lrActualValue,
					fManSyncValue		:= lrManSyncValue,
					bSync				:= bSync,
					eMode				:= eMode,
					bHold				:= bHold,
					stParams			:= stCTRL_PID_PARAMS,
					fOut				=> lrControllerOut,
					bARWactive			=> bARWactive,
					eErrorId			=> eErrorId,
					bError				=> bError
				);

				
// Smooth transition when switching between MANUAL and Auomatic MODE 
IF eMode = eCTRL_MODE_ACTIVE THEN
	lrManSyncValue := lrControllerOut;
END_IF

IF eMode = eCTRL_MODE_MANUAL THEN
	lrSetpointValue := lrActualValue;
END_IF
END_METHOD

METHOD M_Read_Write_Config
VAR_INPUT
END_VAR



IF bEngMode AND bWriteConfig THEN
	
	fbTcConfig.M_WriteConfiguration();
			
ELSIF bEngMode AND bReadConfig THEN
	
	fbTcConfig.M_ReadConfiguration();
		
END_IF



IF NOT fbTcConfig.bIsWriting THEN
	bWriteConfig := FALSE;
END_IF



IF fbTcConfig.bIsReading THEN
	ctrl.lrManualRampUpRate   := cfg.lrRampUpRate;
	ctrl.lrManualRampDownRate := cfg.lrRampDownRate;
ELSIF NOT fbTcConfig.bIsReading THEN
	cfg.lrRampUpRate		:= ctrl.lrManualRampUpRate;
	cfg.lrRampDownRate		:= ctrl.lrManualRampDownRate;
	bReadConfig := FALSE;	
END_IF
END_METHOD

METHOD M_Set_PID_Parameters : BOOL
VAR_INPUT
END_VAR


IF in_bEnable THEN

ctrl.bEnable	:=	TRUE;

END_IF

IF	ctrl.bEnable THEN
	
	stat.bEnabled := TRUE;

	stCTRL_PID_PARAMS.fKp	:= cfg.lrKp;	(* proportional gain Kp	*)
	stCTRL_PID_PARAMS.tTn	:= cfg.tTn;		(*  Integral action time; if this is parameterized to T#0s, the I component is deactivated.								*)
	stCTRL_PID_PARAMS.tTv	:= cfg.tTv;	    (*  Derivative action time; if this is parameterized to T#0s, the D component is deactivated.								*)
	stCTRL_PID_PARAMS.tTd	:= cfg.tTd;	    (*  Damping time								*)
	
	(* set the mode to ACTIVE --> normal operation *)
	eMode					:= eCTRL_MODE_ACTIVE;
	
ELSE
	stat.bEnabled := FALSE;
	eMode					:= eCTRL_MODE_MANUAL;
END_IF
END_METHOD

METHOD M_SetAutoMode
VAR_INPUT
	mode: BOOL;
END_VAR
// AUTO mode can only be activated from MANUAL mode.
// Deactivation is possible only if already in AUTO mode.
IF mode = TRUE	THEN	// Activate AUTO mode
	IF NOT (bAutoMode OR bEngMode)	THEN	// IF MANUAL mode
		bAutoMode := TRUE;	
	END_IF
ELSE	// Deactivate AUTO mode
	IF bAutoMode	THEN	// IF AUTO mode
		bAutoMode := FALSE;	
	END_IF
END_IF
END_METHOD

METHOD M_SetEngMode
VAR_INPUT
	mode: BOOL;
END_VAR
// ENG mode can only be activated from MANUAL mode.
// Deactivation is possible only if already in ENG mode.
// In that case, MANUAL mode will be activated
IF mode = TRUE	THEN	// Activate ENG mode
	IF NOT bAutoMode	THEN	// IF MANUAL mode
		bEngMode := TRUE;	
	END_IF
ELSE	// Deactivate ENG mode
	IF bEngMode	THEN	// IF ENG mode
		bEngMode := FALSE;	
	END_IF
END_IF
END_METHOD

METHOD M_SetManualMode
VAR_INPUT
	cmd: BOOL;
END_VAR
// Manual command can only be set in MANUAL or ENG mode.
// In MANUAL mode, only permitted commands can be set.
IF NOT bAutoMode THEN
	IF bEngMode	THEN
		// ENG mode, any command can be set. No checks!
		bManualMode := cmd;
	ELSE
		// MANUAL mode, only permitted commands can be set.
		//IF (cmd AND bPermitOn) OR (NOT cmd AND bPermitOff)	THEN
			bManualMode := cmd;
		//END_IF
	END_IF
END_IF
END_METHOD

METHOD M_SetPermissionMode : BOOL
VAR_INPUT
END_VAR




IF bAutoMode THEN
	
	stat.sStatus	:= 	'AUTO';
	bManualMode		:=	 FALSE;
	bEngMode		:=	 FALSE;
	
	ctrl.lrRampSetpointValue := in_lrSetPoint;
//	cfg.lrRampUpRate		 := in_lrRampUPRate;
//	cfg.lrRampDownRate		 := in_lrRampDownRate;
	
	// To avaoid abrupt change to the system when changing the Modes
	ctrl.lrManualSetPoint		:= ctrl.lrRampSetpointValue;
	ctrl.lrManualRampUpRate		:= cfg.lrRampUpRate;
	ctrl.lrManualRampDownRate	:= cfg.lrRampDownRate;
ELSIF bEngMode	THEN
	stat.sStatus	:= 'ENG';
	bManualMode		:= FALSE;
	bAutoMode		:= FALSE;
	
	// input from GUI
	M_Read_Write_Config(); (*Read/Write configuration*)
	
	ctrl.lrRampSetpointValue := ctrl.lrManualSetPoint;
	
ELSIF	bManualMode THEN
	stat.sStatus	:= 'MANUAL';
	bAutoMode 		:= FALSE;
	bEngMode		:= FALSE;
	
	// input from GUI
	ctrl.lrRampSetpointValue := ctrl.lrManualSetPoint;


END_IF
END_METHOD

METHOD M_SetRamp : BOOL
VAR_INPUT
//	m_fSetPoint: 			LREAL;
//    m_fRampUPRate:			LREAL;		
//    m_fRampDownRate:		LREAL;
END_VAR

(*Ramp control*)
// TODO: ramp start point should be fActualValue FROM sensor FOR smooth operation

//ctrl.fRampSetpointValue := 		m_fSetPoint;
//ctrl.RampUp_Rate		:=		m_fRampUPRate;					
//ctrl.RampDown_Rate		:=		m_fRampDownRate;			

ramp(in_bEnable := ctrl.bEnable,
			in_fRampSetPoint	:= 	ctrl.lrRampSetpointValue,
			in_fStartPoint		:= 	lrActualValue,
 			in_fRampUp_Rate		:= 	cfg.lrRampUpRate,
 			in_fRampDown_Rate	:= 	cfg.lrRampDownRate,
 			out_fRampValue		=> 	lrSetpointValue);
END_METHOD

END_FUNCTION_BLOCK

// POUs/XML_Cfg_Read_Write/FB_READ_WRITE_TEMP_CONTROL_CONFIG
FUNCTION_BLOCK FB_READ_WRITE_TEMP_CONTROL_CONFIG EXTENDS FB_READ_WRITE_CONFIG_BASE
VAR_INPUT
	in_sTempCtrlName:	T_MaxString;
END_VAR
VAR_IN_OUT
	Temp_Ctrl_Config:   T_METIS_CTRL_BASE_CFG;
END_VAR

SUPER^(
    in_sEntryName  := in_sTempCtrlName,
    in_sSubFolder  := 'Temperature_Control\',
    in_sXPath      := '/Temperature_Control_Configuration/',
    in_pSymAddr    := ADR(Temp_Ctrl_Config),
    in_cbSymSize   := SIZEOF(Temp_Ctrl_Config));

END_FUNCTION_BLOCK

// POUs/Control/Process/FB_FT1_SIM_PROCESS
FUNCTION_BLOCK FB_FT1_SIM_PROCESS
VAR_INPUT
	fIn								: LREAL;
END_VAR
VAR_OUTPUT
	fOut							: LREAL;
END_VAR
VAR
	
	fActualValue					: LREAL;
	fManSyncValue					: LREAL;
	bSync							: BOOL;

	

	eMode							: E_CTRL_MODE;
	stCTRL_PT1_PARAMS				: ST_CTRL_PT1_PARAMS;

	eErrorId						: E_CTRL_ERRORCODES;
	bError							: BOOL;

	(* Filter *)
	fbCTRL_PT1						: FB_CTRL_PT1;

	bInit							: BOOL	:= TRUE;
	fbTON							: TON;
END_VAR

(*-------------------------------------------------------------------*)
(*             PRG_FB_CTRL_PT1_EXAMPLE                  *)
(*-------------------------------------------------------------------*)


IF bInit
THEN
	(* init parameter struct *)
	stCTRL_PT1_PARAMS.tCtrlCycleTime		:= T#10ms;
	stCTRL_PT1_PARAMS.tTaskCycleTime		:= T#10ms;
	stCTRL_PT1_PARAMS.tT1					:= T#1s500ms;
	stCTRL_PT1_PARAMS.fKp					:= 1;

	(* set the mode to ACTIVE --> normal operation *)
	eMode							:= eCTRL_MODE_ACTIVE;

	(* reset the init flag *)
	bInit							:= FALSE;
END_IF

//(* generate input signal *)
//	fbTON(		IN:= TRUE,
//				PT:= T#6s
//			);
//	IF fbTON.Q
//	THEN
//		fbTON(		IN:= FALSE);
//		fIn := -1.0 * fIn;
//	END_IF

(* copy var to scope var *)
//fInToScope := fIn;

(* call filter *)
fbCTRL_PT1(		fIn					:= fIn,
					fManSyncValue	:= fManSyncValue,
					bSync				:= bSync,
					eMode				:= eMode,
					stParams			:= stCTRL_PT1_PARAMS,
					fOut				=> fOut,
					eErrorId			=> eErrorId,
					bError				=> bError
				);


(* copy var to scope var *)
//fOutToScope := fOut;

END_FUNCTION_BLOCK

// POUs/Devices/Heaters/Heater_Ctrl/FB_HEATER_PWM
FUNCTION_BLOCK FB_HEATER_PWM IMPLEMENTS I_Heater
VAR_INPUT
	{attribute 'OPC.UA.DA' := '0'}	
	in_sName:						STRING 	:= 'Heater Controller PWM';	// Controller name
	{attribute 'OPC.UA.DA' := '0'}
	in_fHeaterResistance:			REAL;			// Resistance of the heater to be controlled [Ohms]
	{attribute 'OPC.UA.DA' := '0'}
	in_nMaxHeaterPower:				INT;			// Max power of the heater to be controlled [Ohms]	
	{attribute 'OPC.UA.DA' := '0'}
	in_HeaterCtrlType:				INT 	:= E_METIS_PWM_HEATER_CTRL.Detector_Heater_Ctrl;
	
END_VAR
VAR
	{attribute 'OPC.UA.DA' := '0'}
	nTimeout:					UDINT := 10000;	// Timeout for current to change [ms] after enabling power. Default 10000.
	{attribute 'OPC.UA.DA' := '0'}
	bInterlock:					BOOL := FALSE;	// External Interlock
	{attribute 'OPC.UA.DA' := '0'}
	i_nCouplerState		AT%I*:		UINT;		// Terminal state. Should be 8, i.e. OP.
	
	//{attribute 'OPC.UA.DA' := '0'}
	//q_nSetVoltage		AT%Q*:		INT := 0;	// Adjustable PS voltage [0 - 16383 (0 - 5V)] for liner power supply to power the heater
	//{attribute 'OPC.UA.DA' := '0'}
	//q_nSetCurrent		AT%Q*:		INT := 0;	// Adjustable PS current [0 - 16383 (0 - 4Amps)] for liner power supply to power the heater
 	{attribute 'OPC.UA.DA' := '0'}
	i_nActCurrent		AT%I*:		INT;		// Terminal state. Should be 8, i.e. OP.
	{attribute 'OPC.UA.DA' := '0'}
	i_bReadyToEnable 	AT %I*:		BOOL;
	i_bWarning 			AT %I*: 	BOOL;
	i_bError			AT %I*: 	BOOL;
	i_nDuty_Cycle		AT %I*: 	INT;
	
	
	{attribute 'OPC.UA.DA' := '0'}
	q_bEnable			AT%Q*:		BOOL;		// Enable heater power
	{attribute 'OPC.UA.DA' := '0'}
	q_bEnableDithering	AT %Q* : BOOL := FALSE;
	{attribute 'OPC.UA.DA' := '0'}
	q_bReset			AT %Q* : BOOL;
	{attribute 'OPC.UA.DA' := '0'}
	q_nPWMOut			AT %Q* : INT;			// 
	
	

	stat:		T_METIS_CRYO_HEATER_STATUS;
	ctrl:		T_METIS_CRYO_HEATER_CTRL;

	lrGetPowerVar:		LREAL;
	
	bManualInputFlag:			BOOL := TRUE;
	lrManualHeaterPower:		LREAL := 1.7;
	
	
END_VAR

//IF in_bEnable THEN
//	ctrl.bEnable	:=	TRUE;
//ELSE
//	ctrl.bEnable	:=	FALSE;
//END_IF


IF ctrl.bEnable AND i_bReadyToEnable THEN
	q_bEnable := TRUE;
	stat.bActive := TRUE;
ELSE
	q_bEnable := FALSE;
	stat.bActive := FALSE;
END_IF

//M_Configure();

M_ReadInputs();

M_SetStatus();

M_SetCtrlOutput();

PROPERTY bIsActive : BOOL
GET
bIsActive := stat.bActive;
END_GET
END_PROPERTY

PROPERTY bIsInError : BOOL
GET
bIsInError := stat.bError;
END_GET
END_PROPERTY

PROPERTY bIsNotActive : BOOL
GET
bIsNotActive := NOT stat.bActive;
END_GET
END_PROPERTY

PROPERTY lrHeaterPower : LREAL
GET
lrHeaterPower := ctrl.lrPower;
END_GET
SET
ctrl.lrPower := lrHeaterPower;
END_SET
END_PROPERTY

METHOD M_Activate
VAR_INPUT
END_VAR
ctrl.bEnable := TRUE;
END_METHOD

METHOD M_DeActivate
VAR_INPUT
END_VAR
ctrl.bEnable := FALSE;
END_METHOD

METHOD M_GetHeaterPower : BOOL
VAR_INPUT
	m_lrHeaterPower:  LREAL;
END_VAR
//lrManualHeaterPower := m_lrHeaterPower;

lrGetPowerVar := m_lrHeaterPower;
END_METHOD

METHOD M_ReadInputs
VAR_INPUT
END_VAR
VAR
	m_nActCurrent:		INT;
END_VAR
(*
	Read all inputs and assign values to variables.
*)

m_nActCurrent	:=	i_nActCurrent;

M_ScaleInput(m_nActCurrent:= m_nActCurrent);

// The PWM_Out depends on the Max_current. 
//If the Max current value is correct, 0 - 1000 of m_PWM_Out corresponds to 1 - 100% of duty cycle.  
// (i_nDuty_Cycle/1000) * 100

stat.lrActDutyCycle := (i_nDuty_Cycle/10);

stat.bError 	:= 	i_bError;
stat.bWarning	:=	i_bWarning;
END_METHOD

METHOD M_ScaleInput : BOOL
VAR_INPUT
	m_nActCurrent:	INT;
END_VAR



   

CASE in_HeaterCtrlType OF
	
	E_METIS_PWM_HEATER_CTRL.Detector_Heater_Ctrl:
		// [1 A (rated current)/1024 ] x Actual Current from terminal	
		stat.lrActCurrent :=  (1.0/1024) * m_nActCurrent;	
	
	E_METIS_PWM_HEATER_CTRL.SorptionPump_Heater_Ctrl:
	// [3.5 A (rated current)/1024 ] x Actual Current from terminal	
		stat.lrActCurrent :=  (3.5/1024) * m_nActCurrent;

END_CASE
END_METHOD

METHOD M_ScaleOutput : BOOL
VAR_INPUT
	m_lrCtrlCurrent	:	LREAL;
	m_lrCtrlVoltage	:   LREAL;
END_VAR




////Set PWM 
//q_nSetCurrent := LREAL_TO_INT(m_lrCtrlCurrent / 0.0003051944);

////Set voltage
//// AI from terminal is type INT. Full scale reading (0 - 32767) represent 0 to 10V. 
//// We read only 0 - 5V, so we scale from 0 t 16383 => 5/16383 = 0.0003051944
//// Max Output voltage at 16383 is 60. First translate 0 - 60 into 0 - 5 (5/60 = 0.08333) then 0 - 5 to 0 to 16383
END_METHOD

METHOD M_SetCtrlOutput : BOOL
VAR
	m_lrCtrlPower 	: 	LREAL;
	m_lrCtrlCurrent	:	LREAL;
	m_lrCtrlVoltage	:	LREAL;	 
END_VAR


////Enable the heater
//q_bEnable := ctrl.bEnable;

// Scale power value

//m_lrCtrlPower := 	(ctrl.lrPower/100)*in_nMaxHeaterPower;
////m_lrCtrlPower := 	(in_lrHeaterPower/100)*in_nMaxHeaterPower;


//m_lrCtrlCurrent	:=  SQRT(m_lrCtrlPower/in_nHeaterResistance);

//m_lrCtrlVoltage	:=	SQRT(m_lrCtrlPower * in_nHeaterResistance); 


//M_ScaleOutput(m_lrCtrlCurrent := m_lrCtrlCurrent, m_lrCtrlVoltage := m_lrCtrlVoltage);

// The input % of power is directly related to selecting 0 - 100% PWM_Out duty cycle i.e 32767/100

//IF bManualInputFlag THEN
	//M_SetHeaterPower(M_SetHeaterPower => ctrl.lrPower);
//ELSE
//	ctrl.lrPower := in_lrHeaterPower;
//	lrManualHeaterPower := ctrl.lrPower; // bumpless Mode shift
//END_IF

// Set output to the PWM terminal
q_nPWMOut	:= LREAL_TO_INT(ctrl.lrPower * 327.67);
END_METHOD

METHOD M_SetHeaterPower : LREAL
VAR_INPUT
END_VAR
M_SetHeaterPower := lrGetPowerVar;
END_METHOD

METHOD M_SetManualInputFlag : BOOL
VAR_INPUT
	m_bManual_Input_Flag:		BOOL;
END_VAR
bManualInputFlag := m_bManual_Input_Flag;
END_METHOD

METHOD M_SetStatus : BOOL
VAR_INPUT
END_VAR

// Set actual power I^(Average PWM Voltage)
stat.lrActHeaterPower := ((stat.lrActCurrent * 24 * stat.lrActDutyCycle)/100);

// Set max current
IF in_fHeaterResistance > 0.0 THEN
stat.lrMaxCurrent :=  SQRT(INT_TO_REAL(in_nMaxHeaterPower)/(in_fHeaterResistance));
ELSE
	stat.lrMaxCurrent := 999.9;
END_IF

//IF ctrl.bEnable = TRUE THEN
//	stat.bActive := TRUE;
//ELSE
//	stat.bActive := FALSE;
//END_IF

stat.bHeaterOpenLoop := (stat.lrActCurrent <= 0)
                        AND stat.bActive 
                        AND (ctrl.lrPower > 0);
 
// Check if there is a short circuit: Comparing the actual current with the Max current + 1 A  
 IF stat.lrActCurrent > (stat.lrMaxCurrent + 1) THEN
	 stat.bHeaterShort := TRUE;
 ELSE
	stat.bHeaterShort := FALSE;
 END_IF
 

IF stat.bError THEN
    stat.nHeaterState := E_METIS_CRYO_HEATER_STATE.ERROR;
    stat.sHeaterState := 'ERROR';
ELSIF stat.bActive THEN
    stat.nHeaterState := E_METIS_CRYO_HEATER_STATE.ON;
    stat.sHeaterState := 'ON';
ELSE
    stat.nHeaterState := E_METIS_CRYO_HEATER_STATE.OFF;
    stat.sHeaterState := 'OFF';
END_IF
END_METHOD

END_FUNCTION_BLOCK

// POUs/Devices/Heaters/Heater_Ctrl/I_Heater
INTERFACE I_Heater

PROPERTY bIsActive : BOOL
GET
END_GET
END_PROPERTY

PROPERTY bIsInError : BOOL
GET
END_GET
END_PROPERTY

PROPERTY bIsNotActive : BOOL
GET
END_GET
END_PROPERTY

PROPERTY lrHeaterPower : LREAL
GET
END_GET
SET
END_SET
END_PROPERTY

METHOD M_Activate
VAR_INPUT
END_VAR
END_METHOD

METHOD M_DeActivate
VAR_INPUT
END_VAR
END_METHOD

END_INTERFACE

// POUs/Routines/PowerOutage/FB_METIS_CRYO_POWER_OUTAGE
FUNCTION_BLOCK FB_METIS_CRYO_POWER_OUTAGE
VAR_INPUT
		in_sName:							STRING := 'POWER-OUTAGE';
END_VAR
VAR_OUTPUT
	out_bPowerOutageActive:		BOOL := FALSE;
END_VAR
VAR
	//stat:			T_METIS_CRYO_
		/////////////////////
	// Cryo System logs
	/////////////////////
		
	logs:	FB_CRYO_FUNCTION_LOG;

END_VAR
VAR CONSTANT

    // --- [7000] Preconditions ---
    E7000_InstrumentNotAtNominalTemperature       : UDINT := 7000001; // Instrument not at nominal operation temperature
    E7001_PLCControlNotActive                     : UDINT := 7000002; // PLC control is not active
    E7002_PowerOutageRoutineAlreadyActive         : UDINT := 7000003; // Power outage routine requested while already active
    E7003_SafetyPowerNotAvailable                 : UDINT := 7000004; // Safety power is not available
    E7004_SafetyPowerInsufficient                 : UDINT := 7000005; // Safety power reserve not sufficient for safe-state sequence

    // --- [7100] Detector Protection / Ramp Errors ---
    E7100_DetectorRampTo50KFailed                 : UDINT := 7100001; // Detector ramp to 50 K failed
    E7101_DetectorRampTo90KFailed                 : UDINT := 7100002; // Detector ramp to 90 K failed
    E7102_DetectorRampTooFast                     : UDINT := 7100003; // Detector temperature ramp exceeded allowed rate
    E7103_DetectorTemperatureTooHigh              : UDINT := 7100004; // Detector temperature exceeded allowed limit
    E7104_DetectorTemperatureControlFault         : UDINT := 7100005; // Detector temperature control failed or unstable
    E7105_IMG_NotColdestPointAfter50KRamp         : UDINT := 7100006; // IMG did not become the coldest point after detector ramp to 50 K

    // --- [7200] LN2 / Sorption Pump Protection Errors ---
    E7200_LN2RefillLowerSegmentFailed             : UDINT := 7200001; // Lower segment LN2 refill failed during power outage
    E7201_LN2SupplyNotAvailable                   : UDINT := 7200002; // LN2 supply not available during power outage
    E7202_SorptionPumpTemperatureTooHigh          : UDINT := 7200003; // Sorption pump temperature exceeded allowed limit
    E7203_LN2ValveFailureDuringPowerOutage        : UDINT := 7200004; // LN2 valve failed during power outage sequence
    E7204_LowerSegmentLevelNotRecovered           : UDINT := 7200005; // Lower segment LN2 level did not recover after refill request

    // --- [7300] Safety Power / Timing Errors ---
    E7300_InitialWait10MinFailed                  : UDINT := 7300001; // Initial 10 minute wait phase failed or interrupted
    E7301_5HourHoldPhaseFailed                    : UDINT := 7300002; // 5 hour hold phase failed or interrupted
    E7302_SafeStateSequenceExceeded6Hours         : UDINT := 7300003; // Safe-state sequence exceeded 6 hours
    E7303_SafetyPowerLowBeforeSafeStateCompleted  : UDINT := 7300004; // Safety power became critically low before safe state was reached
    E7304_PowerOutageSequenceTimeout              : UDINT := 7300005; // Overall power outage sequence timed out

    // --- [7400] Temperature Monitoring Errors ---
    E7400_IMG_TemperatureTooHigh                  : UDINT := 7400001; // IMG temperature exceeded allowed limit during power outage handling
    E7401_CFO_TemperatureTooHigh                  : UDINT := 7400002; // CFO temperature exceeded allowed limit during power outage handling
    E7402_DetectorTemperatureSensorFault          : UDINT := 7400003; // Detector temperature sensor invalid or faulty
    E7403_IMGTemperatureSensorFault               : UDINT := 7400004; // IMG temperature sensor invalid or faulty
    E7404_CFOTemperatureSensorFault               : UDINT := 7400005; // CFO temperature sensor invalid or faulty
    E7405_TemperatureTrendUnexpected              : UDINT := 7400006; // Temperature evolution during power outage was unexpected or unsafe

    // --- [7500] Manual Intervention / Recovery ---
    E7500_OperatorAbortedPowerOutageRoutine       : UDINT := 7500001; // Operator manually stopped power outage handling
    E7501_OperatorRestartRequired                 : UDINT := 7500002; // Operator restart required after power outage routine
    E7502_OperatorSelectedInvalidRecoveryMode     : UDINT := 7500003; // Operator selected an invalid operation mode during restart
    E7503_RestartSequenceNotInitiated             : UDINT := 7500004; // Operator did not initiate restart sequence

    // --- [7600] Recovery / Restart Errors ---
    E7600_VacuumPumpsFailedToStart                : UDINT := 7600001; // Vacuum pumps failed to start during recovery
    E7601_AutomaticRefillingFailedToStart         : UDINT := 7600002; // Automatic LN2 refilling failed to start during recovery
    E7602_IMGPrecoolingFailedToStart              : UDINT := 7600003; // IMG precooling failed to start although required
    E7603_CFOPrecoolingFailedToStart              : UDINT := 7600004; // CFO precooling failed to start although required
    E7604_CoolDownRecoveryFailed                  : UDINT := 7600005; // Recovery into cooldown procedure failed
    E7605_PostOutageTemperatureCheckFailed        : UDINT := 7600006; // Temperature validation failed during restart after outage

    // --- [7700] Interlock Violations ---
    E7700_PowerOutageRoutineStartedOutsideNominal : UDINT := 7700001; // Power outage routine started although instrument was not at nominal temperature
    E7701_PLCControlLostDuringPowerOutage         : UDINT := 7700002; // PLC control was lost during power outage routine
    E7702_CoolingCommandIssuedDuringPowerOutage   : UDINT := 7700003; // Cooling command issued during power outage handling
    E7703_UnsafeOperationRequestedDuringOutage    : UDINT := 7700004; // Unsafe operator or software action requested during outage handling

    // --- [7800] Shutdown / Safe-State Failures ---
    E7800_CriticalEquipmentNotInSafeState         : UDINT := 7800001; // Critical equipment could not be placed in safe state
    E7801_DetectorNotInProtectedState             : UDINT := 7800002; // Detector was not left in protected state
    E7802_SorptionPumpNotProtected                : UDINT := 7800003; // Sorption pump was not sufficiently protected
    E7803_PowerOutageSafeStateIncomplete          : UDINT := 7800004; // Safe-state sequence incomplete when routine ended

END_VAR

END_FUNCTION_BLOCK

// POUs/Routines/StopPowerOutage/FB_METIS_CRYO_STOP_POWER_OUTAGE
FUNCTION_BLOCK FB_METIS_CRYO_STOP_POWER_OUTAGE
VAR_INPUT
		in_sName:							STRING := 'STOP-POWER-OUTAGE';
END_VAR
VAR_OUTPUT
	out_bStopPowerOutageActive:		BOOL := FALSE;
END_VAR
VAR
	
	/////////////////////
	// Cryo System logs
	/////////////////////
		
	logs:	FB_CRYO_FUNCTION_LOG;

END_VAR

END_FUNCTION_BLOCK

// POUs/Devices/AmbientPressure/FB_METIS_AMBIENT_PRESSURE_SENSOR
FUNCTION_BLOCK FB_METIS_AMBIENT_PRESSURE_SENSOR EXTENDS FB_CRYO_SENSOR_BASE
VAR_INPUT
	{attribute 'OPC.UA.DA' := '0'}
//	in_nType:	E_CRYO_SENSOR_TYPE_PRESS;
	{attribute 'OPC.UA.DA' := '0'}
	// Scale factor bits -> Volt, U = raw / scale. 
	// Default for 16-bit, +-10V or 0..10V AI: 2^16/10/2 = 3276.8 bit
	in_lrBitsPerVolt:	LREAL := 3276.8;	// Scale factor, U = raw / scale. Default 3276.8
	{attribute 'OPC.UA.DA' := '0'}
	in_nSampleTime:		UINT := 2000;	// Time for average read sample [ms]
END_VAR
VAR_OUTPUT
END_VAR
VAR
	{attribute 'OPC.UA.DA' := '0'}
	stat:	T_CRYO_SENSOR_STATUS_PRESS;	// Complete status

	// Timers 
	{attribute 'OPC.UA.DA' := '0'}
	fbReadTimer:	TON; (* General Timeout *)

	// Misc internal vars
	{attribute 'OPC.UA.DA' := '0'}
	nCount:			UINT := 0;		// Number of effective samples
	{attribute 'OPC.UA.DA' := '0'}
	bReadStarted:	BOOL := FALSE;	// Used for initial trigger of the read timer
	{attribute 'OPC.UA.DA' := '0'}
	lrVoltageSum:	LREAL := 0.0;	// Total sum of Valid voltages during sample time.
	{attribute 'OPC.UA.DA' := '0'}
	lrVoltageAve:	LREAL := 0.0;	// Average voltage over in_nSampleTime
END_VAR

// Set references
RefStat	REF=stat;

IF NOT bReadStarted THEN
	bReadStarted	:= TRUE;
	fbReadTimer(IN:=FALSE);
END_IF
fbReadTimer(IN:=TRUE,PT:=UINT_TO_TIME(in_nSampleTime));


// Execute the base FB
SUPER^();

// Calculate pressure based on the status in input value
METHOD M_SetStatus
VAR_INPUT
END_VAR
VAR
END_VAR
//// Set pressure sensor type
//stat.nType	:= in_nType;

//// Update validity and the pressure in user units, i.e. mbar
//CASE in_nType OF
//	E_CRYO_SENSOR_TYPE_PRESS.PKR_250:
//		M_SetStatus_PKR_250();
//	E_CRYO_SENSOR_TYPE_PRESS.PKR_360:
//		M_SetStatus_PKR_360();
//	E_CRYO_SENSOR_TYPE_PRESS.CMR_361:
//		M_SetStatus_CMR_361();
//	E_CRYO_SENSOR_TYPE_PRESS.WRG_D_NW25:
//		M_SetStatus_WRG_D_NW25();
//END_CASE

M_SetStatus_MIPA_015A();
END_METHOD

// Calculate pressure based on the status in input value
METHOD M_SetStatus_CMR_361
VAR_INPUT
END_VAR
VAR
	// Pfeiffer CMR361 Conversion Volt -> mbar.
	// P = (U - 1) * C1 * C2 [mbar]
	// Defaults are for Pfeiffer CMR361 (note: C1 = 0.125, C2=FullScale = 1000): 
	// P = (U - 1) * 0.125 * 1000.0 = (U-1) * 125[mbar]
	
	lrVoltage:		LREAL;	
END_VAR
// Update validity and the pressure in user units, i.e. mbar.

// Sum up all valid voltages in the range (1.0..9.8V].
IF NOT stat.bInputError  AND  stat.bInputValid  AND stat.bInputActive  THEN
	// Convert bits -> Volt
	lrVoltage	:= i_nValue / in_lrBitsPerVolt;

	// If reading is (1.0..9.8V], add the voltage to the Sum
	IF lrVoltage > 1.0  AND  lrVoltage <= 9.8 THEN
		nCount			:= nCount + 1;
		lrVoltageSum	:= lrVoltageSum + lrVoltage;
	END_IF
END_IF


// If the timer has expired, calculate the average voltage/pressure.
// Also, restart timer, and reset the counter and lrVoltageSum.
IF fbReadTimer.Q THEN
	fbReadTimer(IN:=FALSE);	// Reset timer
	IF nCount > 0 THEN
		stat.lrVoltage	:= lrVoltageSum / nCount;	// Average voltage
	ELSE
		stat.lrVoltage	:= 0.0;	// Dummy voltage - error.
	END_IF
	nCount			:= 0;
	lrVoltageSum	:= 0.0;

	// Convert Volt -> Pressure [mbar]
	// Measuring range [0.1...1100mbar] = [1.0008...9.8V]
	stat.lrPressure		:= (stat.lrVoltage - 1.0) * 125.0;

	// Check the validity of the measurement.
	// < 0.4 V - ERROR, sensor problem, Underrange
	// < 1.0V - NOT Valid, Underrange
	// < 1.0008V (0.1mbar) - Valid, underrange
	//   1.0008V (0.1mbar) .. 9.8V (1100mbar) - Valid, in range
	// > 9.8V (1100mbar) - NOT Valid, Overrange
	IF stat.lrVoltage <= 0.4	THEN
		stat.bError				:= TRUE;
		stat.bValid				:= FALSE;
		stat.bValueInRange		:= FALSE;
		stat.bValueUnderrange	:= TRUE;
		stat.bValueOverrange	:= FALSE;
	ELSIF stat.lrVoltage <= 1.0	THEN
		stat.bError				:= FALSE;
		stat.bValid				:= FALSE;
		stat.bValueInRange		:= FALSE;
		stat.bValueUnderrange	:= TRUE;
		stat.bValueOverrange	:= FALSE;
	ELSIF stat.lrVoltage < 1.0008	THEN
		stat.bError				:= FALSE;
		stat.bValid				:= TRUE;
		stat.bValueInRange		:= FALSE;
		stat.bValueUnderrange	:= TRUE;
		stat.bValueOverrange	:= FALSE;
	ELSIF stat.lrVoltage <= 9.8	THEN
		stat.bError				:= FALSE;
		stat.bValid				:= TRUE;
		stat.bValueInRange		:= TRUE;
		stat.bValueUnderrange	:= FALSE;
		stat.bValueOverrange	:= FALSE;
	ELSE
		stat.bError				:= TRUE;
		stat.bValid				:= FALSE;
		stat.bValueInRange		:= FALSE;
		stat.bValueUnderrange	:= FALSE;
		stat.bValueOverrange	:= TRUE;
	END_IF

END_IF
END_METHOD

METHOD M_SetStatus_MIPA_015A
VAR_INPUT
END_VAR
VAR_INPUT
END_VAR
VAR
    // Honeywell MIP 015P conversion Volt -> pressure (mbar via psi).
    // Ratiometric output: 0.5 ... 4.5 V = 0 ... 15 psi (10 % ... 90 % of Vs)
    // Transfer function (datasheet, ratiometric output):
    //   Vout = 0.8 * Vs * (P - Pmin) / (Pmax - Pmin) + 0.10 * Vs
    // Inverted:
    //   P = (Vout - 0.10 * Vs) * (Pmax - Pmin) / (0.80 * Vs) + Pmin
    //
    // Here: Vs = 5.0 V, Pmin = 0 psi, Pmax = 15 psi.
    // stat.lrPressure will be in mbar (1 psi = 68.947573 mbar).
    
    lrVoltage       : LREAL;
    lrPressurePsi   : LREAL;
    lrPressureMbar  : LREAL;
    lrVs            : LREAL := 5.0;       // Supply voltage [V]
    lrPminPsi       : LREAL := 0.0;       // [psi]
    lrPmaxPsi       : LREAL := 15.0;      // [psi]
    lrSpanPsi       : LREAL;
END_VAR
// Update validity and the pressure in user units, i.e. mbar.
//
// Sum up all valid voltages in the range [0.5 .. 4.5 V].
IF NOT stat.bInputError AND stat.bInputValid AND stat.bInputActive THEN
    // Convert bits -> Volt
    lrVoltage := i_nValue / in_lrBitsPerVolt;

    // If reading is [0.5 .. 4.5 V], add the voltage to the sum for averaging
    IF (lrVoltage >= 0.5) AND (lrVoltage <= 4.5) THEN
        nCount       := nCount + 1;
        lrVoltageSum := lrVoltageSum + lrVoltage;
    END_IF
END_IF

// If the timer has expired, calculate the average voltage/pressure.
// Also, restart timer, and reset the counter and lrVoltageSum.
IF fbReadTimer.Q THEN
    fbReadTimer(IN := FALSE);     // Reset timer

    IF nCount > 0 THEN
        stat.lrVoltage := lrVoltageSum / nCount;    // Average voltage
    ELSE
        stat.lrVoltage := 0.0;                      // Dummy voltage - error.
    END_IF

    nCount       := 0;
    lrVoltageSum := 0.0;

    // --- Convert Volt -> Pressure ---
    // Use only if Vs is valid and voltage within a reasonable range.
    lrSpanPsi := lrPmaxPsi - lrPminPsi;             // = 15 psi

    IF (lrVs > 0.0) THEN
        // Compute pressure in psi from the averaged voltage
        lrPressurePsi := (stat.lrVoltage - (0.10 * lrVs)) * lrSpanPsi / (0.80 * lrVs) + lrPminPsi;

        // Clamp to physical range [0 .. 15 psi]
        IF lrPressurePsi < lrPminPsi THEN
            lrPressurePsi := lrPminPsi;
        ELSIF lrPressurePsi > lrPmaxPsi THEN
            lrPressurePsi := lrPmaxPsi;
        END_IF;

        // Convert psi -> mbar
        lrPressureMbar := lrPressurePsi * 68.947573;

        // Default assignment; may be overwritten for overrange cases below
        stat.lrPressure := lrPressureMbar;
    ELSE
        // Invalid Vs -> cannot compute meaningful pressure
        lrPressurePsi   := 0.0;
        lrPressureMbar  := 0.0;
        stat.lrPressure := 0.0;
    END_IF

    // --- Check the validity of the measurement based on voltage ---
    // Diagnostic rails (datasheet, ratiometric output):
    //   ~0.125 V (2.5 % Vs) and ~4.875 V (97.5 % Vs) for internal error/overpressure.
    //
    // Here we use the following ranges:
    //   <= 0.125 V or >= 4.875 V : Error (sensor fault / severe over/under condition)
    //   < 0.5 V                  : Not valid, underrange
    //   0.5 V .. 4.5 V           : Valid, in range
    //   > 4.5 V and < 4.875 V    : Valid, overrange (pressure clamped to max)
    IF stat.lrVoltage <= 0.125 THEN
        // Sensor internal failure or severe underrange
        stat.bError             := TRUE;
        stat.bValid             := FALSE;
        stat.bValueInRange      := FALSE;
        stat.bValueUnderrange   := TRUE;
        stat.bValueOverrange    := FALSE;
        stat.lrPressure         := 0.0;

    ELSIF stat.lrVoltage < 0.5 THEN
        // Underrange: below normal transfer function region
        stat.bError             := FALSE;
        stat.bValid             := FALSE;
        stat.bValueInRange      := FALSE;
        stat.bValueUnderrange   := TRUE;
        stat.bValueOverrange    := FALSE;
        stat.lrPressure         := 0.0;

    ELSIF stat.lrVoltage <= 4.5 THEN
        // Normal operating range: 0 .. 15 psi
        stat.bError             := FALSE;
        stat.bValid             := TRUE;
        stat.bValueInRange      := TRUE;
        stat.bValueUnderrange   := FALSE;
        stat.bValueOverrange    := FALSE;
        // stat.lrPressure already set from transfer function.

    ELSIF stat.lrVoltage < 4.875 THEN
        // Overrange but below diagnostic rail: clamp to full-scale (15 psi)
        stat.bError             := FALSE;
        stat.bValid             := TRUE;
        stat.bValueInRange      := FALSE;
        stat.bValueUnderrange   := FALSE;
        stat.bValueOverrange    := TRUE;
        stat.lrPressure         := lrPmaxPsi * 68.947573;  // 15 psi -> mbar

    ELSE
        // At or above diagnostic rail: treat as error / severe overpressure
        stat.bError             := TRUE;
        stat.bValid             := FALSE;
        stat.bValueInRange      := FALSE;
        stat.bValueUnderrange   := FALSE;
        stat.bValueOverrange    := TRUE;
        stat.lrPressure         := lrPmaxPsi * 68.947573;  // keep at max as a safe value
    END_IF

END_IF
END_METHOD

// Calculate pressure based on the status in input value
METHOD M_SetStatus_PKR_250
VAR_INPUT
END_VAR
VAR
	// Pfeiffer PKR250/251 Conversion Volt -> mbar.
	// P = 10^(C1 * U - C2).
	// Defaults are for Pfeiffer PKR250/251 (note: C1 = 1.667, C2 = d = 11.33): 
	// P = 10^(1.667 * U - 11.33)
	// Valid range for U is 1.8-8.6
	//
	
	lrVoltage:		LREAL;
END_VAR
// Update validity and the pressure in user units, i.e. mbar.

// Sum up all valid voltages in the range [1.4..9.5V].
IF NOT stat.bInputError  AND  stat.bInputValid  AND stat.bInputActive  THEN
	// Convert bits -> Volt
	lrVoltage	:= i_nValue / in_lrBitsPerVolt;

	// If reading is [1.4..9.5V], add the voltage to the Sum
	IF lrVoltage >= 1.4  AND  lrVoltage <= 9.5 THEN
		nCount			:= nCount + 1;
		lrVoltageSum	:= lrVoltageSum + lrVoltage;
	END_IF
END_IF


// If the timer has expired, calculate the average voltage/pressure.
// Also, restart timer, and reset the counter and lrVoltageSum.
IF fbReadTimer.Q THEN
	fbReadTimer(IN:=FALSE);	// Reset timer
	IF nCount > 0 THEN
		stat.lrVoltage	:= lrVoltageSum / nCount;	// Average voltage
	ELSE
		stat.lrVoltage	:= 0.0;	// Dummy voltage - error.
	END_IF
	nCount			:= 0;
	lrVoltageSum	:= 0.0;

	// Convert Volt -> Pressure [mbar]
	// Measuring range [0.1...1100mbar] = [1.0008...9.8V]
	stat.lrPressure		:= EXPT(10.0, (1.667 * stat.lrVoltage - 11.33));

	// Check the validity of the measurement.
	// < 0.5 V - ERROR, sensor problem, Underrange
	// < 1.4V (1E-09mbar)- NOT Valid, Underrange
	// < 1.76V (4E-09mbar) - Valid, underrange
	//   1.76V (4E-09mbar) .. 8.6V (1014mbar) - Valid, in range
	// < 9.5V (1014mbar) - Valid, Overrange, fixed pressure to 1014mbar
	// >= 9.5V  - NOT Valid, Overrange
	IF stat.lrVoltage <= 0.5	THEN
		stat.bError				:= TRUE;
		stat.bValid				:= FALSE;
		stat.bValueInRange		:= FALSE;
		stat.bValueUnderrange	:= TRUE;
		stat.bValueOverrange	:= FALSE;
	ELSIF stat.lrVoltage < 1.4	THEN
		stat.bError				:= FALSE;
		stat.bValid				:= FALSE;
		stat.bValueInRange		:= FALSE;
		stat.bValueUnderrange	:= TRUE;
		stat.bValueOverrange	:= FALSE;
	ELSIF stat.lrVoltage < 1.76	THEN
		stat.bError				:= FALSE;
		stat.bValid				:= TRUE;
		stat.bValueInRange		:= FALSE;
		stat.bValueUnderrange	:= TRUE;
		stat.bValueOverrange	:= FALSE;
	ELSIF stat.lrVoltage <= 8.6	THEN
		stat.bError				:= FALSE;
		stat.bValid				:= TRUE;
		stat.bValueInRange		:= TRUE;
		stat.bValueUnderrange	:= FALSE;
		stat.bValueOverrange	:= FALSE;
	ELSIF stat.lrVoltage <= 9.5	THEN
		stat.bError				:= FALSE;
		stat.bValid				:= TRUE;
		stat.bValueInRange		:= FALSE;
		stat.bValueUnderrange	:= FALSE;
		stat.bValueOverrange	:= TRUE;
		stat.lrPressure			:= 1014.0;
	ELSE
		stat.bError				:= TRUE;
		stat.bValid				:= FALSE;
		stat.bValueInRange		:= FALSE;
		stat.bValueUnderrange	:= FALSE;
		stat.bValueOverrange	:= TRUE;
	END_IF

END_IF
END_METHOD

// Calculate pressure based on the status in input value
METHOD M_SetStatus_PKR_360
VAR_INPUT
END_VAR
VAR
	// Pfeiffer PKR360 Conversion Volt -> mbar.
	// P = 10^(C1 * U - C2).
	// Defaults are for Pfeiffer PKR250/251 (note: C1 = 1.667, C2 = d = 11.33): 
	// P = 10^(1.667 * U - 11.33)
	// Valid range for U is 1.397-8.6 (up to 9.5 fixed to 1014 mbar in SW)
	//
	
	lrVoltage:		LREAL;
END_VAR
// Update validity and the pressure in user units, i.e. mbar.

// Sum up all valid voltages in the range [1.397 .. 9.5V].
IF NOT stat.bInputError  AND  stat.bInputValid  AND stat.bInputActive  THEN
	// Convert bits -> Volt
	lrVoltage	:= i_nValue / in_lrBitsPerVolt;

	// If reading is [1.4..9.5V], add the voltage to the Sum
	IF lrVoltage >= 1.397  AND  lrVoltage <= 9.5 THEN
		nCount			:= nCount + 1;
		lrVoltageSum	:= lrVoltageSum + lrVoltage;
	END_IF
END_IF


// If the timer has expired, calculate the average voltage/pressure.
// Also, restart timer, and reset the counter and lrVoltageSum.
IF fbReadTimer.Q THEN
	fbReadTimer(IN:=FALSE);	// Reset timer
	IF nCount > 0 THEN
		stat.lrVoltage	:= lrVoltageSum / nCount;	// Average voltage
	ELSE
		stat.lrVoltage	:= 0.0;	// Dummy voltage - error.
	END_IF
	nCount			:= 0;
	lrVoltageSum	:= 0.0;

	// Convert Volt -> Pressure [mbar]
	// Measuring range [0.1...1100mbar] = [1.0008...9.5V]
	stat.lrPressure		:= EXPT(10.0, (1.667 * stat.lrVoltage - 11.33));

	// Check the validity of the measurement.
	// < 1.217 V - ERROR, sensor problem, Underrange
	// < 1.397V (1E-09mbar)- NOT Valid, Underrange
	//   8.6V (4E-09mbar) .. 8.6V (1014mbar) - Valid, in range
	// < 9.5V (1014mbar) - Valid, Overrange, fixed pressure to 1014mbar
	// >= 9.5V  - NOT Valid, Overrange
	IF stat.lrVoltage <= 1.217	THEN
		stat.bError				:= TRUE;
		stat.bValid				:= FALSE;
		stat.bValueInRange		:= FALSE;
		stat.bValueUnderrange	:= TRUE;
		stat.bValueOverrange	:= FALSE;
	ELSIF stat.lrVoltage < 1.397	THEN
		stat.bError				:= FALSE;
		stat.bValid				:= FALSE;
		stat.bValueInRange		:= FALSE;
		stat.bValueUnderrange	:= TRUE;
		stat.bValueOverrange	:= FALSE;
	ELSIF stat.lrVoltage <= 8.6	THEN
		stat.bError				:= FALSE;
		stat.bValid				:= TRUE;
		stat.bValueInRange		:= TRUE;
		stat.bValueUnderrange	:= FALSE;
		stat.bValueOverrange	:= FALSE;
	ELSIF stat.lrVoltage <= 9.5	THEN
		stat.bError				:= FALSE;
		stat.bValid				:= TRUE;
		stat.bValueInRange		:= FALSE;
		stat.bValueUnderrange	:= FALSE;
		stat.bValueOverrange	:= TRUE;
		stat.lrPressure			:= 1014.0;
	ELSE
		stat.bError				:= TRUE;
		stat.bValid				:= FALSE;
		stat.bValueInRange		:= FALSE;
		stat.bValueUnderrange	:= FALSE;
		stat.bValueOverrange	:= TRUE;
	END_IF

END_IF
END_METHOD

// Calculate pressure based on the status in input value
METHOD M_SetStatus_WRG_D_NW25
VAR_INPUT
END_VAR
VAR
	// Edwards WRG-D-NW25 Conversion Volt -> mbar.
	// Range 10^-9 .. 100
	// P = 10^(C1 * U - C2).
	// P = 10^(1.5 * U - 12.0)
	// Valid range for U is 2.0-10.0
	//
	
	lrVoltage:		LREAL;
END_VAR
// Update validity and the pressure in user units, i.e. mbar.

// Sum up all valid voltages in the range [2.0..10.0V].
IF NOT stat.bInputError  AND  stat.bInputValid  AND stat.bInputActive  THEN
	// Convert bits -> Volt
	lrVoltage	:= i_nValue / in_lrBitsPerVolt;

	// If reading is [2.0..10.0V], add the voltage to the Sum
	IF lrVoltage >= 2.0  AND  lrVoltage <= 10.0 THEN
		nCount			:= nCount + 1;
		lrVoltageSum	:= lrVoltageSum + lrVoltage;
	END_IF
END_IF


// If the timer has expired, calculate the average voltage/pressure.
// Also, restart timer, and reset the counter and lrVoltageSum.
IF fbReadTimer.Q THEN
	fbReadTimer(IN:=FALSE);	// Reset timer
	IF nCount > 0 THEN
		stat.lrVoltage	:= lrVoltageSum / nCount;	// Average voltage
	ELSE
		stat.lrVoltage	:= 0.0;	// Dummy voltage - error.
	END_IF
	nCount			:= 0;
	lrVoltageSum	:= 0.0;

	// Convert Volt -> Pressure [mbar]
	// Measuring range [0.1...1000mbar] = [2.0...10.0V]
	stat.lrPressure		:= EXPT(10.0, (1.5 * stat.lrVoltage - 12.0));

	// Check the validity of the measurement.
	// < 1.5 V - ERROR, sensor problem, Underrange
	// < 2.0V (1E-09mbar)- NOT Valid, Underrange
	// < 10.0V (1000mbar) - Valid
	// < 10.15V (1678mbar) - NOT Valid, Overrange
	// >= 10.15V  - Error, Overrange
	IF stat.lrVoltage < 1.5	THEN
		stat.bError				:= TRUE;
		stat.bValid				:= FALSE;
		stat.bValueInRange		:= FALSE;
		stat.bValueUnderrange	:= TRUE;
		stat.bValueOverrange	:= FALSE;
	ELSIF stat.lrVoltage < 2.0	THEN
		stat.bError				:= FALSE;
		stat.bValid				:= FALSE;
		stat.bValueInRange		:= FALSE;
		stat.bValueUnderrange	:= TRUE;
		stat.bValueOverrange	:= FALSE;
	ELSIF stat.lrVoltage <= 10.0	THEN
		stat.bError				:= FALSE;
		stat.bValid				:= TRUE;
		stat.bValueInRange		:= TRUE;
		stat.bValueUnderrange	:= FALSE;
		stat.bValueOverrange	:= FALSE;
	ELSIF stat.lrVoltage <= 10.15	THEN
		stat.bError				:= FALSE;
		stat.bValid				:= FALSE;
		stat.bValueInRange		:= FALSE;
		stat.bValueUnderrange	:= FALSE;
		stat.bValueOverrange	:= TRUE;
	ELSE
		stat.bError				:= TRUE;
		stat.bValid				:= FALSE;
		stat.bValueInRange		:= FALSE;
		stat.bValueUnderrange	:= FALSE;
		stat.bValueOverrange	:= TRUE;
	END_IF

END_IF
END_METHOD

END_FUNCTION_BLOCK

// POUs/Simulation/FB_SIM_VENTING_VALVES
FUNCTION_BLOCK FB_SIM_VENTING_VALVES
VAR
	//	// Output valve control signals
	i_bON_N2V_1	AT %I*:	BOOL;
	i_bON_N2V_2	AT %I*:	BOOL;
	
	// Simulation of ON/open feedback signal
	q_bON_N2V_1	AT %Q*:	BOOL := FALSE;
	q_bON_N2V_2	AT %Q*:	BOOL := FALSE;
	
	// Simulation of OFF/closed feedback signal
	q_bOFF_N2V_1	AT %Q*:	BOOL := TRUE;
	q_bOFF_N2V_2	AT %Q*:	BOOL := TRUE;
	
	q_nCouplerState	AT %Q*:	INT := 8;
END_VAR

// Valve Simulation 

// ON signals are active low
q_bON_N2V_1	:= i_bON_N2V_1;
q_bON_N2V_2	:= i_bON_N2V_2;


// OFF signals are active low
q_bOFF_N2V_1	:= NOT i_bON_N2V_1;
q_bOFF_N2V_2	:= NOT i_bON_N2V_2;

END_FUNCTION_BLOCK

// POUs/Simulation/FB_SIM_PRE_COOLING_VALVES
FUNCTION_BLOCK FB_SIM_PRE_COOLING_VALVES
VAR
	//	// Output valve control signals
	i_bON_PVV_P1	AT %I*:	BOOL;
	i_bON_PVV_P2	AT %I*:	BOOL;
	i_bON_PVV_P3	AT %I*:	BOOL;
	
	
	// Simulation of ON/open feedback signal
	q_bON_PVV_P1	AT %Q*:	BOOL := FALSE;
	q_bON_PVV_P2	AT %Q*:	BOOL := FALSE;
	q_bON_PVV_P3	AT %Q*:	BOOL := FALSE;
	
	
	// Simulation of OFF/closed feedback signal
	q_bOFF_PVV_P1	AT %Q*:	BOOL := TRUE;
	q_bOFF_PVV_P2	AT %Q*:	BOOL := TRUE;
	q_bOFF_PVV_P3	AT %Q*:	BOOL := TRUE;
	
	
	q_nCouplerState	AT %Q*:	INT := 8;
END_VAR

// Valve Simulation 

// ON signals are active low
//q_bON_N2V_1	:= i_bON_N2V_1;

q_bON_PVV_P1	:= i_bON_PVV_P1;
q_bON_PVV_P2	:= i_bON_PVV_P2;
q_bON_PVV_P3	:= i_bON_PVV_P3;


// OFF signals are active low
//q_bOFF_N2V_1	:= NOT i_bON_N2V_1;

q_bOFF_PVV_P1	:= NOT i_bON_PVV_P1;
q_bOFF_PVV_P2	:= NOT i_bON_PVV_P2;
q_bOFF_PVV_P3	:= NOT i_bON_PVV_P3;

END_FUNCTION_BLOCK

// POUs/Simulation/FB_SIM_LN2_SENSOR
FUNCTION_BLOCK FB_SIM_LN2_SENSOR
VAR_INPUT
END_VAR
VAR_OUTPUT
END_VAR
VAR
	
	q_nStatus_HA	AT%Q*:	UINT	:= 0;	// Simulated status
	q_nValue_HA	    AT%Q*:	INT		:= -211;	// Simulated value [bit]
	
	q_nStatus_H		AT%Q*:	UINT	:= 0;	// Simulated status
	q_nValue_H		AT%Q*:	INT		:= -211;	// Simulated value [bit]
	
	q_nStatus_L		AT%Q*:	UINT	:= 0;	// Simulated status
	q_nValue_L		AT%Q*:	INT		:= -211;	// Simulated value [bit]
	
	q_nStatus_LA	AT%Q*:	UINT	:= 0;	// Simulated status
	q_nValue_LA 	AT%Q*:	INT		:= -2111;	// Simulated value [bit]
	
	i_bSensorHeaters	AT%I*:	BOOL;		
	
	
END_VAR

END_FUNCTION_BLOCK

// POUs/Simulation/FB_SIM_LN2_LEVEL_VALVES
FUNCTION_BLOCK FB_SIM_LN2_LEVEL_VALVES
VAR
	//	// Output valve control signals
	i_bON_SHA_V		AT %I*:	BOOL;
	i_bON_SHB_V		AT %I*:	BOOL;
	i_bON_SHC_V		AT %I*:	BOOL;
	
	// Simulation of ON/open feedback signal
	q_bON_SHA_V		AT %Q*:	BOOL := FALSE;
	q_bON_SHB_V		AT %Q*:	BOOL := FALSE;
	q_bON_SHC_V		AT %Q*:	BOOL := FALSE;
	
	// Simulation OF OFF/closed feedback signal
	q_bOFF_SHA_V	AT %Q*:	BOOL := TRUE;
	q_bOFF_SHB_V	AT %Q*:	BOOL := TRUE;
	q_bOFF_SHC_V	AT %Q*:	BOOL := TRUE;
	
	q_nCouplerState	AT %Q*:	INT := 8;
END_VAR

// Valve Simulation 

// ON signals are active low
q_bON_SHA_V	:= i_bON_SHA_V;
q_bON_SHB_V	:= i_bON_SHB_V;
q_bON_SHC_V	:= i_bON_SHC_V;

// OFF signals are active low
q_bOFF_SHA_V	:= NOT i_bON_SHA_V;
q_bOFF_SHB_V	:= NOT i_bON_SHB_V;
q_bOFF_SHC_V	:= NOT i_bON_SHC_V;

END_FUNCTION_BLOCK

// POUs/Simulation/FB_SIM_REGENERATION
FUNCTION_BLOCK FB_SIM_REGENERATION
VAR_INPUT
END_VAR
VAR_OUTPUT
END_VAR
VAR
	sim_ReadyToEnable	AT %Q*:		BOOL := TRUE;
	sim_t_sp_1			AT %Q*:		REAL := 100.0;
	sim_t_sp_2			AT %Q*:		REAL := 100.0;
	
	temp_ramp_1: FB_CTRL_RAMP_GENERATOR;
	temp_ramp_2: FB_CTRL_RAMP_GENERATOR;
	
	
	bEnable_Ramp: BOOL := TRUE;
	
	stParams: ST_CTRL_RAMP_GENERATOR_PARAMS := (tTaskCycleTime := T#10MS, tCtrlCycleTime := T#10MS, fVeloPos := 0.03, fVeloNeg := 0.030);
	
	sim_h_sp_bError AT %Q*:		BOOL := FALSE;
	sim_h_sp_bWarning AT %Q*:		BOOL := FALSE;
	
	sim_sp_heater_current : LREAL := 0.25;
	
	sim_sp_nActCurrent AT %Q* : DINT;
	
END_VAR



//temp_ramp_1(
//	bEnable:= bEnable_Ramp, 
//	fStart:= 260, 
//	fTarget:= 330, 
//	fOut=> sim_t_sp_1, 
//	fVeloOut=> , 
//	bValueReached=> , 
//	eErrorId=> , 
//	bError=> , 
//	stParams:= stParams);
	
	
//temp_ramp_1(
//	bEnable:= bEnable_Ramp, 
//	fStart:= 260, 
//	fTarget:= 330, 
//	fOut=> sim_t_sp_2, 
//	fVeloOut=> , 
//	bValueReached=> , 
//	eErrorId=> , 
//	bError=> , 
//	stParams:= stParams);

sim_t_sp_1 := sim_t_sp_1 + 0.0001;
sim_t_sp_2 := sim_t_sp_2 + 0.0001;
			

sim_sp_nActCurrent := LREAL_TO_DINT((sim_sp_heater_current/3.5) * 1024);

END_FUNCTION_BLOCK

// POUs/Devices/Heaters/Heater_Ctrl/FB_METIS_HEATER
FUNCTION_BLOCK FB_METIS_HEATER
VAR_INPUT
    {attribute 'OPC.UA.DA' := '0'}
	{attribute 'TcHmiSymbol.Show'}
	{attribute 'TcHmiSymbol.ReadOnly'}    
    in_sName:               STRING  := 'Heater'; // Heater name
    {attribute 'OPC.UA.DA' := '0'}
	{attribute 'TcHmiSymbol.Show'}
	{attribute 'TcHmiSymbol.ReadOnly'}
    in_lrHeaterResistance:  LREAL;               // Resistance of the heater to be controlled [Ohms]
    {attribute 'OPC.UA.DA' := '0'}
	{attribute 'TcHmiSymbol.Show'}
	{attribute 'TcHmiSymbol.ReadOnly'}
    in_lrHeaterMaxPower:    LREAL;               // Max power of the heater to be controlled [Watts]    
    {attribute 'OPC.UA.DA' := '0'}
	{attribute 'TcHmiSymbol.Show'}
	{attribute 'TcHmiSymbol.ReadOnly'}
    in_eHeaterType:         E_METIS_CRYO_HEATER_TYPE := E_METIS_CRYO_HEATER_TYPE.NONE;
    {attribute 'OPC.UA.DA' := '0'}
    in_sAutoSetpointSource:     STRING;          // Name of the source of the AUTO setpoint
    {attribute 'OPC.UA.DA' := '0'}
    in_lrAutoSetpointValue:     LREAL;           // Output power coming for the AUTO setpoint
END_VAR
VAR
    {attribute 'OPC.UA.DA' := '0'}
    nTimeout:                   UDINT := 10000;     // Timeout for current to change [ms] after enabling power. Default 10000.
    {attribute 'OPC.UA.DA' := '0'}
    bInterlock:                 BOOL := FALSE;      // External Interlock
    {attribute 'OPC.UA.DA' := '0'}
    i_nCouplerState     AT %I*: UINT;               // Terminal state. Should be 8, i.e. OP.
    
    {attribute 'OPC.UA.DA' := '0'}
    io_pwm      : T_METIS_HEATER_IO_PWM;
    {attribute 'OPC.UA.DA' := '0'}
    io_cpau60   : T_METIS_HEATER_IO_CPAU60;
    {attribute 'OPC.UA.DA' := '0'}
    io_cxwui60  : T_METIS_HEATER_IO_CXWUI60;
    {attribute 'OPC.UA.DA' := '0'}
    io_el95x1   : T_METIS_HEATER_IO_EL95X1;
    
    {attribute 'OPC.UA.DA' := '1'}
	{attribute 'TcHmiSymbol.Show'}
    stat:        T_METIS_HEATER_STAT;
    {attribute 'OPC.UA.DA' := '1'}
	{attribute 'TcHmiSymbol.Show'}
    ctrl:        T_METIS_HEATER_CTRL;
    {attribute 'OPC.UA.DA' := '1'}
	{attribute 'TcHmiSymbol.Show'}
    cfg:         T_METIS_HEATER_CFG;

    {attribute 'OPC.UA.DA' := '0'}
	{attribute 'TcHmiSymbol.Show'}
    fbConfig    : FB_READ_WRITE_HEATER_CONFIG; 
	
	tonThermalSwitchOpen : TON;
    
    // some temporary variables to experiment with
    rEl95x1HysteresisLowRange : REAL := 3;  // below 3V, switch range to LOW RANGE
    rEl95x1HysteresisHighRange : REAL := 4;  // below 4V, switch range to HIGH RANGE
    rEl95x1HysteresisDisable : REAL := 0.2;  // below 0.2V, fully disconnect the heater (e.g. with a relay)
    rEl95x1HysteresisEnable : REAL := 0.3;  // above 0.3V, fully connect the heater (e.g. with a relay)
	
			// Alarm handling
	// List of alarms to be handled by Temperature
	arrEventEntry : ARRAY [0..4] OF TcEventEntry;
	// Alarm handler FB
	fbAlarmHandler : FB_AlarmHandler;
	{attribute 'TcHmiSymbol.Show'}
	{attribute 'TcHmiSymbol.ReadOnly'}
	sInstanceName : T_MaxString;
	{attribute 'TcHmiSymbol.Show'}
	bConfirmAllAlarms : BOOL;
	{attribute 'TcHmiSymbol.Show'}
	{attribute 'TcHmiSymbol.ReadOnly'}
	sEventClassName : T_MaxString;
	
	// Logs logs
	logs:	FB_CRYO_FUNCTION_LOG;
    
    
END_VAR

IF not stat.bConfigured THEN
    M_Configure();
END_IF

// Read/write the configuration
fbConfig(in_sHeaterName:= in_sName, cfg := cfg);

M_SetMode();

M_SetEnable();

M_ReadInputs();

M_SetStatus();

M_SetCtrlOutput();

// read/write the config (if needed)
M_Read_Write_Config();


// Handle alarms
M_UpdateAlarms();

METHOD M_Configure
VAR_INPUT
END_VAR
VAR_INST
    {attribute 'OPC.UA.DA' := '0'}
    nConfigureState : INT;
END_VAR
arrEventEntry[0] := Tc_Events.METISCryoHeaterEventClass.HeaterShortCircuit;
arrEventEntry[1] := Tc_Events.METISCryoHeaterEventClass.HeaterOpenCircuit;
arrEventEntry[2] := Tc_Events.METISCryoHeaterEventClass.HeaterManualMode;
arrEventEntry[3] := Tc_Events.METISCryoHeaterEventClass.HeaterThermalSwitchOpen;
arrEventEntry[4] := Tc_Events.METISCryoHeaterEventClass.HeaterInsufficientPower;

CASE nConfigureState OF
    0:  
        // set some defaults
        stat.eCtrlMode := E_METIS_CTRL_MODE.AUTO;   // always start in AUTO mode
        cfg.lrAutoScalePercent := 100.0;            // 100% by default
        
        // start reading the config
        fbConfig.M_ReadConfiguration();
        nConfigureState := 1;
    1:
        IF fbConfig.bReadingDoneFlag THEN
            
            // clear the flag
            fbConfig.M_ClearReadingDoneFlag();
            
            // set the bConfigured flag
            stat.bConfigured := TRUE;

        END_IF
END_CASE
END_METHOD

METHOD M_isHeaterInError : BOOL
VAR_INPUT
END_VAR
M_isHeaterInError := stat.bError;
END_METHOD

METHOD M_Read_Write_Config
VAR_INPUT
END_VAR
VAR_IN_OUT
END_VAR

IF ctrl.bWriteConfig THEN
    
    // (update the cfg object if needed)
    // ...
    
    // write the cfg object
    fbConfig.M_WriteConfiguration();
    ctrl.bWriteConfig := FALSE;
            
ELSIF ctrl.bReadConfig THEN

    fbConfig.M_ReadConfiguration();
    ctrl.bReadConfig := FALSE;
    
END_IF


IF fbConfig.bReadingDoneFlag THEN
    // clear the flag
    fbConfig.M_ClearReadingDoneFlag();
END_IF
END_METHOD

METHOD M_ReadInputs
VAR_INPUT
END_VAR
VAR
END_VAR
(*
    Read all inputs and assign values to variables.
*)

CASE in_eHeaterType OF
    
    E_METIS_CRYO_HEATER_TYPE.PWM_DETECTOR,
    E_METIS_CRYO_HEATER_TYPE.PWM_SORPTION,
    E_METIS_CRYO_HEATER_TYPE.PWM_WINDOW:
        M_ScaleInput(m_nActCurrent:= io_pwm.i_nActCurrent);
        
        // The PWM_Out depends on the Max_current. 
        // If the Max current value is correct, 0 - 1000 of m_PWM_Out corresponds to 1 - 100% of duty cycle.  
        // (i_nDuty_Cycle/1000) * 100
        stat.lrActDutyCycle := INT_TO_LREAL(io_pwm.i_nDuty_Cycle)/10.0;
        stat.bActDutyCycleAvailable := TRUE;
        
        stat.bHwError     := io_pwm.i_bError;
        stat.bHwWarning   := io_pwm.i_bWarning;

    E_METIS_CRYO_HEATER_TYPE.CPAU60:
        M_ScaleInput(m_nActCurrent:= io_cpau60.i_nActCurrent);
        stat.bActDutyCycleAvailable := FALSE;

    E_METIS_CRYO_HEATER_TYPE.CXWUI60:
        M_ScaleInput(m_nActCurrent:= io_cxwui60.i_nActCurrent);
        stat.bActDutyCycleAvailable := FALSE;

    E_METIS_CRYO_HEATER_TYPE.EL95X1:
    
        IF io_el95x1.q_bEnable THEN
            stat.lrActCurrent := REAL_TO_LREAL(io_el95x1.i_rCurrent);
            stat.lrActVoltage := REAL_TO_LREAL(io_el95x1.i_rVoltage);
        ELSE
            stat.lrActCurrent := 0;
            stat.lrActVoltage := 0;
        END_IF
        
        stat.bHwError     := io_el95x1.i_bError;
        stat.bHwWarning   := io_el95x1.i_bWarning;
        
        stat.bActDutyCycleAvailable := FALSE;

END_CASE
END_METHOD

METHOD M_ScaleInput : BOOL
VAR_INPUT
    m_nActCurrent:    DINT;
END_VAR
   

CASE in_eHeaterType OF
    
    E_METIS_CRYO_HEATER_TYPE.PWM_DETECTOR:
        // [1 A (rated current)/1024 ] x Actual Current from terminal    
        stat.lrActCurrent :=  (1.0/1024) * DINT_TO_LREAL(m_nActCurrent);    
    
    E_METIS_CRYO_HEATER_TYPE.PWM_SORPTION,
    E_METIS_CRYO_HEATER_TYPE.PWM_WINDOW:
        // [3.5 A (rated current)/1024 ] x Actual Current from terminal    
        stat.lrActCurrent :=  (3.5/1024) * DINT_TO_LREAL(m_nActCurrent);

    E_METIS_CRYO_HEATER_TYPE.CPAU60:
        (* EL3681 Digital Multimeter terminal
        
            Scaled presentation:
            corresponds to 1 bit per µV / µA,
            Examples:
             Mode 0, Autorange, 2.5 V: 2,500,000 decimal
             Mode 2, 800 mA: 800,000 decimal 
        *) 
        stat.lrActCurrent :=  DINT_TO_LREAL(m_nActCurrent) / 1000000.0; 

    E_METIS_CRYO_HEATER_TYPE.CXWUI60:
        // AI from terminal is type INT. Full scale reading (0 - 32767) represent 0 to 10V. 
        // We read only 0 - 5V, so we scale from 0 t 16383 => 5/16383 = 0.0003051944
        stat.lrActCurrent :=  DINT_TO_LREAL(m_nActCurrent) * 0.0003051944; 

END_CASE
END_METHOD

METHOD M_ScaleOutput : BOOL
VAR_INPUT
    m_lrCtrlCurrent    :    LREAL;
    m_lrCtrlVoltage    :   LREAL;
END_VAR


CASE in_eHeaterType OF
    
    E_METIS_CRYO_HEATER_TYPE.PWM_DETECTOR,
    E_METIS_CRYO_HEATER_TYPE.PWM_SORPTION,
    E_METIS_CRYO_HEATER_TYPE.PWM_WINDOW:
        // no current to set (only PWMout)
        ;

    E_METIS_CRYO_HEATER_TYPE.CPAU60:
        
        // Set voltage
        // AI from terminal is type INT. Full scale reading (0 - 32767) represent 0 to 10V. 
        // We read 0 - 10V, so we scale from 0 t 32767 => 10/32767 =  0.00030518509
        // Max Output voltage at 16383 is 60. First translate 0 - 60 into 0 - 10 (10/60 = 0.166666 ) then 0 - 10 to 0 to 32767
        io_cpau60.q_nSetVoltage := LREAL_TO_INT( (m_lrCtrlVoltage * 0.166666) / 0.00030518509);

    E_METIS_CRYO_HEATER_TYPE.CXWUI60:
                
        //Set current 
        io_cxwui60.q_nSetCurrent  := LREAL_TO_INT(m_lrCtrlCurrent / 0.0003051944);
        
        // Set voltage
        // AI from terminal is type INT. Full scale reading (0 - 32767) represent 0 to 10V. 
        // We read only 0 - 5V, so we scale from 0 t 16383 => 5/16383 = 0.0003051944
        // Max Output voltage at 16383 is 60. First translate 0 - 60 into 0 - 5 (5/60 = 0.08333) then 0 - 5 to 0 to 16383
        io_cxwui60.q_nSetVoltage := LREAL_TO_INT( (m_lrCtrlVoltage * 0.08333) / 0.0003051944 );

    E_METIS_CRYO_HEATER_TYPE.EL95X1:
        // set voltage
        io_el95x1.q_rSetVoltage := LREAL_TO_REAL(m_lrCtrlVoltage);
        
        // apply some histeresis on the range switching:
        //   if setpoint > 4V -> switch to high ramge (13)
        //   if setpoint < 3V -> switch to low range (15)
        IF m_lrCtrlVoltage > rEl95x1HysteresisHighRange AND io_el95x1.q_nOutputInterface <> 13 THEN
            io_el95x1.q_nOutputInterface := 13;
        ELSIF m_lrCtrlVoltage < rEl95x1HysteresisLowRange AND io_el95x1.q_nOutputInterface <> 15 THEN
            io_el95x1.q_nOutputInterface := 15;
        END_IF
         
        
END_CASE
END_METHOD

METHOD M_SetCtrlOutput : BOOL
VAR
	lrCtrlPower 	: 	LREAL;
	lrCtrlCurrent	:	LREAL;
	lrCtrlVoltage	:	LREAL;	 
END_VAR
CASE in_eHeaterType OF
    
    E_METIS_CRYO_HEATER_TYPE.PWM_DETECTOR:

        lrCtrlPower := 	(stat.lrActSetpoint / 100.0) * in_lrHeaterMaxPower;
        lrCtrlCurrent := SQRT(lrCtrlPower / in_lrHeaterResistance); // in Amps
        
        io_pwm.q_nPWMOut :=  LREAL_TO_INT(lrCtrlCurrent * 32767 / 1.0);
        
    E_METIS_CRYO_HEATER_TYPE.PWM_SORPTION,
    E_METIS_CRYO_HEATER_TYPE.PWM_WINDOW:
    
        lrCtrlPower := 	(stat.lrActSetpoint / 100.0) * in_lrHeaterMaxPower;
        lrCtrlCurrent := SQRT(lrCtrlPower / in_lrHeaterResistance); // in Amps
        
        io_pwm.q_nPWMOut :=  LREAL_TO_INT(lrCtrlCurrent * 32767 / 3.5);
        
        //io_pwm.q_nPWMOut := LREAL_TO_INT(stat.lrActSetpoint * 327.67);

    E_METIS_CRYO_HEATER_TYPE.CPAU60:
        
        lrCtrlPower := 	(stat.lrActSetpoint / 100.0) * in_lrHeaterMaxPower;
        lrCtrlCurrent	:=  SQRT(lrCtrlPower / in_lrHeaterResistance);
        lrCtrlVoltage	:=	SQRT(lrCtrlPower * in_lrHeaterResistance); 
        
        M_ScaleOutput(m_lrCtrlCurrent := lrCtrlCurrent, m_lrCtrlVoltage := lrCtrlVoltage);

    E_METIS_CRYO_HEATER_TYPE.CXWUI60:
        
        lrCtrlPower   := stat.lrActSetpoint / 100.0 * in_lrHeaterMaxPower;
        lrCtrlCurrent	:= SQRT(lrCtrlPower / in_lrHeaterResistance);
        lrCtrlVoltage	:= SQRT(lrCtrlPower * in_lrHeaterResistance); 
        
        M_ScaleOutput(m_lrCtrlCurrent := lrCtrlCurrent, m_lrCtrlVoltage := lrCtrlVoltage);

    E_METIS_CRYO_HEATER_TYPE.EL95X1:
        lrCtrlPower   := stat.lrActSetpoint / 100.0 * in_lrHeaterMaxPower;
        lrCtrlVoltage	:= SQRT(lrCtrlPower * in_lrHeaterResistance); 
        
        M_ScaleOutput(m_lrCtrlCurrent := 0 (* not used *), m_lrCtrlVoltage := lrCtrlVoltage);
        
END_CASE
END_METHOD

METHOD M_SetDisable
VAR_INPUT
END_VAR

IF stat.bAuto THEN
    stat.bActive := FALSE;
ELSIF stat.bManual THEN
    stat.bActive := ctrl.bManualEnable;
END_IF

CASE in_eHeaterType OF
    E_METIS_CRYO_HEATER_TYPE.PWM_DETECTOR, 
    E_METIS_CRYO_HEATER_TYPE.PWM_SORPTION, 
    E_METIS_CRYO_HEATER_TYPE.PWM_WINDOW:
        stat.bActive := stat.bActive AND io_pwm.i_bReadyToEnable;
        io_pwm.q_bEnable := stat.bActive;
    E_METIS_CRYO_HEATER_TYPE.CPAU60:
	    io_cpau60.q_bEnable := stat.bActive;
    E_METIS_CRYO_HEATER_TYPE.CXWUI60:
	    io_cxwui60.q_bEnable := stat.bActive;
    E_METIS_CRYO_HEATER_TYPE.EL95X1:
        IF stat.bActive THEN
            // 0.2V is the minimum that the EL95X1 can deliver
            // So, below this setpoint, we fully disconnect the power, but we apply some hysteresis:
            //     setpoint < 0.2V -> OFF
            //     setpoint > 0.3V -> ON 
            
            // the heater should be ON above the hysteresis threshold
            IF io_el95x1.q_rSetVoltage > rEl95x1HysteresisEnable AND (NOT io_el95x1.q_bEnable) THEN
                io_el95x1.q_bEnable := TRUE; 
            // the heater should be OFF below the hysteresis threshold
            ELSIF io_el95x1.q_rSetVoltage < rEl95x1HysteresisDisable AND io_el95x1.q_bEnable THEN
                io_el95x1.q_bEnable := FALSE;
			END_IF
        ELSE
            io_el95x1.q_bEnable := FALSE; 
        END_IF
        
        IF io_el95x1.q_bEnable THEN
            io_el95x1.q_nOutputOperation := 1;
        ELSE
            io_el95x1.q_nOutputOperation := 0;
		END_IF
END_CASE
END_METHOD

METHOD M_SetEnable
VAR_INPUT
END_VAR

IF stat.bAuto THEN
    stat.bActive := TRUE;
ELSIF stat.bManual THEN
    stat.bActive := ctrl.bManualEnable;
END_IF

CASE in_eHeaterType OF
    E_METIS_CRYO_HEATER_TYPE.PWM_DETECTOR, 
    E_METIS_CRYO_HEATER_TYPE.PWM_SORPTION, 
    E_METIS_CRYO_HEATER_TYPE.PWM_WINDOW:
        stat.bActive := stat.bActive AND io_pwm.i_bReadyToEnable;
        // We put q_bEnable to FALSE when the setpoint is 0.00 (i.e. below 0.01) 
        // because of an issue found at IMG/SCA subsystem testing: at setpoint 0.00 %
        // there are still some milliamps of current flowing if q_bEnable is TRUE!
        io_pwm.q_bEnable := stat.bActive AND stat.lrActSetpoint >= 0.009;
    E_METIS_CRYO_HEATER_TYPE.CPAU60:
	    io_cpau60.q_bEnable := stat.bActive;
    E_METIS_CRYO_HEATER_TYPE.CXWUI60:
	    io_cxwui60.q_bEnable := stat.bActive;
    E_METIS_CRYO_HEATER_TYPE.EL95X1:
        IF stat.bActive THEN
            // 0.2V is the minimum that the EL95X1 can deliver
            // So, below this setpoint, we fully disconnect the power, but we apply some hysteresis:
            //     setpoint < 0.2V -> OFF
            //     setpoint > 0.3V -> ON 
            
            // the heater should be ON above the hysteresis threshold
            IF io_el95x1.q_rSetVoltage > rEl95x1HysteresisEnable AND (NOT io_el95x1.q_bEnable) THEN
                io_el95x1.q_bEnable := TRUE; 
            // the heater should be OFF below the hysteresis threshold
            ELSIF io_el95x1.q_rSetVoltage < rEl95x1HysteresisDisable AND io_el95x1.q_bEnable THEN
                io_el95x1.q_bEnable := FALSE;
			END_IF
        ELSE
            io_el95x1.q_bEnable := FALSE; 
        END_IF
        
        IF io_el95x1.q_bEnable THEN
            io_el95x1.q_nOutputOperation := 1;
        ELSE
            io_el95x1.q_nOutputOperation := 0;
		END_IF
        
END_CASE
END_METHOD

METHOD M_SetMode
VAR_INPUT
END_VAR
If stat.eCtrlMode = E_METIS_CTRL_MODE.NONE THEN
    // typical behavior when e.g. a config file did not contain a valid entry
    // To avoid problems, force MANUAL in this case
    stat.eCtrlMode := E_METIS_CTRL_MODE.MANUAL;
END_IF

// check which mode switches are accepted
// (currently very simple, but can be made more complex if needed)
stat.bAcceptCtrlMode_Auto := stat.eCtrlMode = E_METIS_CTRL_MODE.MANUAL
                             AND NOT stat.bError;
stat.bAcceptCtrlMode_Manual := stat.eCtrlMode = E_METIS_CTRL_MODE.AUTO ;

// switch to AUTO / MANUAL mode if acceptable
IF ctrl.eCtrlMode = E_METIS_CTRL_MODE.AUTO AND stat.bAcceptCtrlMode_Auto THEN
    stat.eCtrlMode := E_METIS_CTRL_MODE.AUTO;
ELSIF ctrl.eCtrlMode = E_METIS_CTRL_MODE.MANUAL AND stat.bAcceptCtrlMode_Manual THEN
    stat.eCtrlMode := E_METIS_CTRL_MODE.MANUAL;
END_IF

// update the redundant booleans (for easy HMI development)
stat.bAuto   := stat.eCtrlMode = E_METIS_CTRL_MODE.AUTO;
stat.bManual := stat.eCtrlMode = E_METIS_CTRL_MODE.MANUAL;

// update the actual setpoint
IF stat.bAuto THEN
    stat.lrActSetpoint := in_lrAutoSetpointValue * LIMIT(0, cfg.lrAutoScalePercent, 100) / 100.0;
ELSIF stat.bManual THEN
    stat.lrActSetpoint := ctrl.lrManualSetpoint;
ELSE
    stat.lrActSetpoint := 0.0;
END_IF

// reset any request
ctrl.eCtrlMode := E_METIS_CTRL_MODE.NONE;
END_METHOD

METHOD M_SetStatus : BOOL
VAR_INPUT
END_VAR
VAR
    lrExpectedPower             : LREAL;
    lrPowerRatio                : LREAL;
    bThermalSwitchOpenCandidate : BOOL;
END_VAR
M_SetStatus := FALSE;

sInstanceName := fbAlarmHandler.sInstanceName;
sEventClassName := fbAlarmHandler.sEventClassName;
IF bConfirmAllAlarms THEN
	bConfirmAllAlarms := FALSE;
	fbAlarmHandler.M_ConfirmAllAlarms();
END_IF


stat.lrAutoCtrlOut := in_lrAutoSetpointValue;

(*
lrPowerRatio < 0.10  -> open circuit
0.10 <= lrPowerRatio < 0.85 -> thermal switch open
high demand + low power -> insufficient heater power
*)

// ----------------------------------------------------
// Calculate actual heater power
// ----------------------------------------------------
CASE in_eHeaterType OF

    E_METIS_CRYO_HEATER_TYPE.PWM_DETECTOR,
    E_METIS_CRYO_HEATER_TYPE.PWM_WINDOW:
        // I²R
        stat.lrActHeaterPower :=
            stat.lrActCurrent * stat.lrActCurrent * in_lrHeaterResistance;

    E_METIS_CRYO_HEATER_TYPE.PWM_SORPTION:
        // Approximate PWM power: I * Vavg
        stat.lrActHeaterPower :=
            stat.lrActCurrent * 24.0 * stat.lrActDutyCycle / 100.0;

    E_METIS_CRYO_HEATER_TYPE.CPAU60:
        // I²R
        stat.lrActHeaterPower :=
            stat.lrActCurrent * stat.lrActCurrent * in_lrHeaterResistance;

    E_METIS_CRYO_HEATER_TYPE.CXWUI60:
        // I²R
        stat.lrActHeaterPower :=
            stat.lrActCurrent * stat.lrActCurrent * in_lrHeaterResistance;

    E_METIS_CRYO_HEATER_TYPE.EL95X1:
        IF stat.bActive THEN
            stat.lrActHeaterPower := stat.lrActCurrent * stat.lrActVoltage;
        ELSE
            stat.lrActHeaterPower := 0.0;
        END_IF;

ELSE
    stat.lrActHeaterPower := 0.0;

END_CASE;


